C01818=1103.978,373.015,-89.633,-179.779,17.252,151.645
C01819=1103.984,373.262,-89.668,-179.776,17.255,151.645
C01820=1103.989,373.509,-89.704,-179.773,17.259,151.646
C01821=1103.995,373.757,-89.740,-179.770,17.264,151.646
C01822=1104.002,374.004,-89.776,-179.768,17.268,151.646
C01823=1104.007,374.251,-89.811,-179.765,17.272,151.647
C01824=1104.012,374.499,-89.848,-179.762,17.276,151.647
C01825=1104.018,374.745,-89.884,-179.760,17.280,151.648
C01826=1104.024,374.993,-89.919,-179.757,17.284,151.648
C01827=1104.029,375.240,-89.955,-179.754,17.289,151.649
C01828=1104.035,375.487,-89.992,-179.751,17.293,151.649
C01829=1104.041,375.735,-90.028,-179.748,17.297,151.650
C01830=1104.046,375.982,-90.064,-179.746,17.302,151.650
C01831=1104.052,376.229,-90.100,-179.743,17.306,151.651
C01832=1104.058,376.476,-90.135,-179.740,17.310,151.651
C01833=1104.063,376.724,-90.172,-179.737,17.314,151.652
C01834=1104.069,376.971,-90.208,-179.735,17.319,151.653
C01835=1104.075,377.218,-90.244,-179.732,17.323,151.653
C01836=1104.080,377.466,-90.281,-179.728,17.328,151.653
C01837=1104.086,377.713,-90.316,-179.727,17.332,151.654
C01838=1104.092,377.960,-90.352,-179.724,17.336,151.655
C01839=1104.097,378.208,-90.389,-179.721,17.341,151.655
C01840=1104.103,378.454,-90.425,-179.718,17.345,151.656
C01841=1104.108,378.702,-90.461,-179.716,17.349,151.656
C01842=1104.115,378.949,-90.498,-179.713,17.354,151.657
C01843=1104.120,379.195,-90.534,-179.710,17.358,151.657
C01844=1104.126,379.443,-90.570,-179.707,17.363,151.658
C01845=1104.132,379.690,-90.606,-179.704,17.368,151.659
C01846=1104.137,379.938,-90.643,-179.702,17.372,151.659
C01847=1104.143,380.185,-90.679,-179.699,17.376,151.660
C01848=1104.149,380.432,-90.716,-179.696,17.381,151.660
C01849=1104.155,380.680,-90.752,-179.694,17.385,151.661
C01850=1104.160,380.927,-90.788,-179.691,17.390,151.661
C01851=1104.166,381.174,-90.825,-179.689,17.394,151.662
C01852=1104.171,381.422,-90.861,-179.686,17.399,151.663
C01853=1104.178,381.669,-90.897,-179.683,17.404,151.663
C01854=1104.183,381.915,-90.934,-179.680,17.408,151.664
C01855=1104.189,382.162,-90.971,-179.678,17.413,151.664
C01856=1104.195,382.410,-91.008,-179.674,17.417,151.665
C01857=1104.201,382.657,-91.043,-179.673,17.422,151.666
C01858=1104.210,383.071,-91.105,-179.668,17.430,151.667
C01859=1104.219,383.485,-91.166,-179.663,17.438,151.668
C01860=1104.228,383.899,-91.227,-179.659,17.446,151.669
C01861=1104.239,384.314,-91.289,-179.655,17.454,151.670
C01862=1104.244,384.561,-91.326,-179.652,17.458,151.671
C01863=1104.249,384.808,-91.363,-179.649,17.463,151.671
C01864=1104.256,385.055,-91.399,-179.647,17.468,151.672
C01865=1104.261,385.302,-91.436,-179.644,17.473,151.673
C01866=1104.266,385.549,-91.473,-179.641,17.478,151.673
C01867=1104.273,385.796,-91.509,-179.639,17.483,151.674
C01868=1104.278,386.043,-91.546,-179.636,17.488,151.675
C01869=1104.284,386.291,-91.583,-179.634,17.493,151.676
C01870=1104.289,386.537,-91.620,-179.631,17.498,151.676
C01871=1104.295,386.785,-91.657,-179.629,17.502,151.677
C01872=1104.301,387.032,-91.694,-179.626,17.507,151.678
C01873=1104.306,387.279,-91.731,-179.624,17.512,151.678
C01874=1104.312,387.526,-91.768,-179.621,17.517,151.679
C01875=1104.318,387.773,-91.805,-179.619,17.522,151.680
C01876=1104.324,388.020,-91.841,-179.616,17.527,151.681
C01877=1104.329,388.267,-91.879,-179.613,17.532,151.681
C01878=1104.335,388.514,-91.916,-179.611,17.537,151.682
C01879=1104.340,388.762,-91.953,-179.609,17.542,151.683
C01880=1104.346,389.009,-91.990,-179.606,17.547,151.684
C01881=1104.353,389.256,-92.027,-179.603,17.552,151.684
C01882=1104.358,389.503,-92.064,-179.601,17.557,151.685
C01883=1104.364,389.750,-92.101,-179.598,17.563,151.686
C01884=1104.369,389.996,-92.138,-179.596,17.568,151.687
C01885=1104.375,390.244,-92.175,-179.593,17.573,151.687
C01886=1104.380,390.491,-92.212,-179.591,17.578,151.688
C01887=1104.386,390.738,-92.250,-179.588,17.583,151.689
C01888=1104.393,390.985,-92.287,-179.586,17.588,151.690
C01889=1104.398,391.232,-92.324,-179.583,17.593,151.690
C01890=1104.404,391.479,-92.361,-179.581,17.599,151.691
C01891=1104.410,391.726,-92.398,-179.578,17.604,151.692
C01892=1104.415,391.974,-92.435,-179.576,17.609,151.693
C01893=1104.421,392.220,-92.473,-179.573,17.615,151.694
C01894=1104.427,392.468,-92.510,-179.570,17.620,151.695
C01895=1104.433,392.715,-92.548,-179.568,17.625,151.695
C01896=1104.438,392.962,-92.585,-179.565,17.631,151.696
C01897=1104.444,393.209,-92.623,-179.563,17.636,151.697
C01898=1104.450,393.456,-92.660,-179.561,17.641,151.698
C01899=1104.456,393.703,-92.698,-179.558,17.646,151.699
C01900=1104.461,393.950,-92.735,-179.556,17.652,151.700
C01901=1104.467,394.197,-92.772,-179.553,17.657,151.701
C01902=1104.473,394.444,-92.809,-179.551,17.663,151.702
C01903=1104.479,394.691,-92.847,-179.549,17.668,151.703
C01904=1104.483,394.939,-92.885,-179.547,17.673,151.703
C01905=1104.489,395.185,-92.923,-179.544,17.679,151.704
C01906=1104.495,395.432,-92.960,-179.541,17.685,151.705
C01907=1104.501,395.680,-92.997,-179.539,17.690,151.706
C01908=1104.507,395.926,-93.035,-179.537,17.696,151.707
C01909=1104.513,396.173,-93.073,-179.534,17.701,151.708
C01910=1104.518,396.387,-93.105,-179.533,17.706,151.709
C01911=1104.523,396.600,-93.138,-179.530,17.711,151.709
C01912=1104.528,396.813,-93.170,-179.529,17.716,151.710
C01913=1104.533,397.026,-93.203,-179.526,17.721,151.711
C01914=1104.537,397.239,-93.236,-179.524,17.725,151.712
C01915=1104.542,397.453,-93.269,-179.522,17.731,151.713
C01916=1104.547,397.666,-93.301,-179.520,17.735,151.714
C01917=1104.552,397.879,-93.334,-179.518,17.741,151.714
C01918=1104.557,398.126,-93.371,-179.516,17.746,151.715
C01919=1104.563,398.373,-93.408,-179.513,17.752,151.716
C01920=1104.569,398.621,-93.447,-179.511,17.757,151.717
C01921=1104.575,398.868,-93.485,-179.509,17.763,151.718
C01922=1104.581,399.114,-93.523,-179.506,17.769,151.719
C01923=1104.586,399.361,-93.560,-179.504,17.775,151.720
C01924=1104.592,399.608,-93.599,-179.502,17.781,151.721
C01925=1104.597,399.855,-93.636,-179.500,17.786,151.722
C01926=1104.604,400.103,-93.674,-179.497,17.793,151.723
C01927=1104.609,400.350,-93.712,-179.495,17.798,151.724
C01928=1104.615,400.597,-93.750,-179.493,17.804,151.725
C01929=1104.620,400.844,-93.788,-179.491,17.810,151.727
C01930=1104.626,401.090,-93.826,-179.488,17.816,151.728
C01931=1104.631,401.338,-93.864,-179.486,17.822,151.729
C01932=1104.638,401.585,-93.902,-179.484,17.828,151.730
C01933=1104.643,401.832,-93.940,-179.482,17.834,151.731
C01934=1104.649,402.079,-93.979,-179.479,17.840,151.732
C01935=1104.655,402.326,-94.016,-179.477,17.846,151.733
C01936=1104.660,402.573,-94.055,-179.475,17.852,151.734
C01937=1104.666,402.820,-94.093,-179.472,17.859,151.735
C01938=1104.671,403.067,-94.131,-179.470,17.865,151.736
C01939=1104.678,403.313,-94.170,-179.468,17.871,151.737
C01940=1104.683,403.560,-94.208,-179.465,17.877,151.738
C01941=1104.689,403.808,-94.246,-179.463,17.883,151.739
C01942=1104.694,404.055,-94.284,-179.462,17.889,151.741
C01943=1104.700,404.302,-94.322,-179.459,17.896,151.742
C01944=1104.706,404.549,-94.361,-179.457,17.902,151.743
C01945=1104.712,404.796,-94.400,-179.455,17.908,151.744
C01946=1104.717,405.042,-94.438,-179.453,17.915,151.745
C01947=1104.723,405.290,-94.476,-179.451,17.921,151.746
C01948=1104.729,405.537,-94.514,-179.448,17.928,151.748
C01949=1104.735,405.783,-94.553,-179.446,17.933,151.749
C01950=1104.740,406.030,-94.592,-179.444,17.940,151.750
C01951=1104.746,406.277,-94.629,-179.442,17.946,151.751
C01952=1104.752,406.524,-94.669,-179.440,17.953,151.752
C01953=1104.757,406.771,-94.707,-179.437,17.960,151.754
C01954=1104.763,407.018,-94.745,-179.435,17.965,151.755
C01955=1104.769,407.265,-94.784,-179.433,17.972,151.756
C01956=1104.774,407.512,-94.823,-179.431,17.979,151.757
C01957=1104.780,407.758,-94.861,-179.429,17.986,151.758
C01958=1104.786,408.006,-94.900,-179.427,17.992,151.760
C01959=1104.791,408.253,-94.938,-179.424,17.999,151.761
C01960=1104.797,408.500,-94.977,-179.423,18.005,151.762
C01961=1104.802,408.747,-95.016,-179.420,18.012,151.763
C01962=1104.809,408.994,-95.055,-179.418,18.018,151.765
C01963=1104.814,409.241,-95.093,-179.416,18.026,151.766
C01964=1104.820,409.488,-95.132,-179.414,18.032,151.767
C01965=1104.825,409.735,-95.171,-179.412,18.039,151.769
C01966=1104.830,409.948,-95.205,-179.410,18.045,151.770
C01967=1104.835,410.161,-95.238,-179.408,18.051,151.771
C01968=1104.840,410.374,-95.272,-179.407,18.056,151.772
C01969=1104.845,410.587,-95.304,-179.405,18.062,151.773
C01970=1104.849,410.800,-95.338,-179.403,18.068,151.774
C01971=1104.854,411.013,-95.372,-179.401,18.074,151.775
C01972=1104.860,411.226,-95.405,-179.399,18.080,151.776
C01973=1104.864,411.439,-95.439,-179.398,18.086,151.778
C01974=1104.869,411.686,-95.478,-179.395,18.093,151.779
C01975=1104.876,411.933,-95.517,-179.393,18.100,151.780
C01976=1104.882,412.179,-95.556,-179.392,18.107,151.782
C01977=1104.888,412.426,-95.595,-179.389,18.114,151.783
C01978=1104.893,412.673,-95.633,-179.387,18.121,151.784
C01979=1104.899,412.921,-95.673,-179.385,18.128,151.786
C01980=1104.905,413.167,-95.712,-179.383,18.135,151.787
C01981=1104.911,413.414,-95.751,-179.381,18.142,151.789
C01982=1104.916,413.661,-95.790,-179.379,18.149,151.790
C01983=1104.922,413.908,-95.829,-179.377,18.156,151.791
C01984=1104.927,414.155,-95.868,-179.375,18.164,151.793
C01985=1104.933,414.402,-95.908,-179.374,18.171,151.794
C01986=1104.939,414.648,-95.947,-179.371,18.178,151.796
C01987=1104.945,414.896,-95.986,-179.369,18.185,151.797
C01988=1104.950,415.142,-96.025,-179.367,18.193,151.799
C01989=1104.956,415.389,-96.065,-179.365,18.200,151.800
C01990=1104.962,415.636,-96.104,-179.363,18.207,151.802
C01991=1104.968,415.883,-96.143,-179.361,18.215,151.803
C01992=1104.973,416.129,-96.182,-179.359,18.222,151.804
C01993=1104.980,416.376,-96.222,-179.358,18.229,151.806
C01994=1104.985,416.623,-96.261,-179.355,18.236,151.807
C01995=1104.991,416.870,-96.300,-179.353,18.244,151.809
C01996=1104.996,417.117,-96.340,-179.351,18.252,151.810
C01997=1105.002,417.364,-96.379,-179.349,18.259,151.812
C01998=1105.007,417.610,-96.418,-179.348,18.267,151.814
C01999=1105.014,417.857,-96.458,-179.346,18.274,151.815
C02000=1105.019,418.103,-96.498,-179.344,18.282,151.817
C02001=1105.025,418.351,-96.538,-179.342,18.290,151.818
C02002=1105.031,418.598,-96.577,-179.340,18.297,151.820
C02003=1105.036,418.844,-96.616,-179.338,18.305,151.821
C02004=1105.042,419.091,-96.656,-179.336,18.313,151.823
C02005=1105.047,419.337,-96.696,-179.334,18.321,151.825
C02006=1105.053,419.584,-96.735,-179.333,18.328,151.826
C02007=1105.059,419.831,-96.774,-179.331,18.336,151.828
C02008=1105.065,420.077,-96.815,-179.329,18.344,151.830
C02009=1105.071,420.325,-96.855,-179.327,18.352,151.831
C02010=1105.076,420.571,-96.894,-179.325,18.360,151.833
C02011=1105.082,420.818,-96.934,-179.323,18.368,151.834
C02012=1105.087,421.065,-96.973,-179.321,18.375,151.836
C02013=1105.093,421.312,-97.013,-179.319,18.383,151.838
C02014=1105.100,421.558,-97.053,-179.318,18.392,151.839
C02015=1105.104,421.805,-97.093,-179.316,18.400,151.841
C02016=1105.111,422.051,-97.133,-179.314,18.408,151.843
C02017=1105.117,422.299,-97.172,-179.312,18.416,151.844
C02018=1105.122,422.545,-97.213,-179.310,18.424,151.846
C02019=1105.128,422.792,-97.252,-179.308,18.432,151.848
C02020=1105.134,423.038,-97.292,-179.307,18.440,151.850
C02021=1105.139,423.285,-97.332,-179.305,18.448,151.851
C02022=1105.144,423.505,-97.368,-179.304,18.455,151.853
C02023=1105.150,423.724,-97.403,-179.302,18.463,151.854
C02024=1105.155,423.944,-97.439,-179.300,18.470,151.856
C02025=1105.160,424.164,-97.474,-179.299,18.477,151.858
C02026=1105.164,424.383,-97.510,-179.297,18.485,151.859
C02027=1105.169,424.604,-97.546,-179.296,18.492,151.861
C02028=1105.174,424.822,-97.582,-179.294,18.500,151.862
C02029=1105.179,425.043,-97.618,-179.293,18.507,151.864
C02030=1105.186,425.289,-97.658,-179.291,18.516,151.866
C02031=1105.191,425.536,-97.697,-179.290,18.524,151.868
C02032=1105.197,425.782,-97.738,-179.288,18.533,151.869
C02033=1105.203,426.029,-97.778,-179.286,18.542,151.871
C02034=1105.208,426.275,-97.818,-179.284,18.550,151.873
C02035=1105.214,426.523,-97.858,-179.282,18.559,151.875
C02036=1105.220,426.769,-97.898,-179.281,18.567,151.877
C02037=1105.226,427.016,-97.939,-179.279,18.576,151.879
C02038=1105.231,427.262,-97.979,-179.278,18.584,151.881
C02039=1105.237,427.509,-98.020,-179.277,18.593,151.883
C02040=1105.243,427.755,-98.060,-179.274,18.602,151.885
C02041=1105.249,428.002,-98.100,-179.273,18.611,151.886
C02042=1105.254,428.249,-98.140,-179.271,18.619,151.888
C02043=1105.260,428.495,-98.181,-179.270,18.628,151.890
C02044=1105.266,428.742,-98.221,-179.268,18.637,151.892
C02045=1105.272,428.989,-98.262,-179.266,18.646,151.894
C02046=1105.277,429.236,-98.302,-179.265,18.655,151.896
C02047=1105.283,429.481,-98.342,-179.263,18.664,151.898
C02048=1105.289,429.728,-98.383,-179.262,18.673,151.900
C02049=1105.294,429.975,-98.424,-179.260,18.682,151.902
C02050=1105.300,430.221,-98.465,-179.259,18.691,151.904
C02051=1105.306,430.467,-98.505,-179.257,18.700,151.906
C02052=1105.312,430.714,-98.546,-179.255,18.710,151.908
C02053=1105.317,430.961,-98.586,-179.254,18.719,151.910
C02054=1105.323,431.208,-98.627,-179.253,18.728,151.912
C02055=1105.329,431.454,-98.668,-179.251,18.737,151.914
C02056=1105.334,431.700,-98.708,-179.249,18.747,151.917
C02057=1105.340,431.946,-98.749,-179.248,18.756,151.919
C02058=1105.346,432.193,-98.790,-179.247,18.765,151.921
C02059=1105.352,432.440,-98.831,-179.245,18.775,151.923
C02060=1105.357,432.687,-98.871,-179.244,18.784,151.925
C02061=1105.363,432.933,-98.913,-179.243,18.793,151.927
C02062=1105.368,433.179,-98.953,-179.241,18.803,151.929
C02063=1105.375,433.426,-98.993,-179.240,18.812,151.931
C02064=1105.381,433.672,-99.035,-179.238,18.822,151.934
C02065=1105.386,433.919,-99.076,-179.237,18.832,151.936
C02066=1105.392,434.166,-99.116,-179.236,18.841,151.938
C02067=1105.398,434.412,-99.158,-179.234,18.851,151.940
C02068=1105.403,434.659,-99.198,-179.233,18.861,151.943
C02069=1105.408,434.904,-99.240,-179.231,18.870,151.945
C02070=1105.414,435.151,-99.281,-179.230,18.880,151.947
C02071=1105.419,435.398,-99.322,-179.229,18.890,151.949
C02072=1105.425,435.644,-99.363,-179.228,18.900,151.951
C02073=1105.431,435.891,-99.404,-179.226,18.910,151.954
C02074=1105.437,436.137,-99.445,-179.225,18.919,151.956
C02075=1105.443,436.384,-99.487,-179.224,18.930,151.958
C02076=1105.448,436.630,-99.528,-179.223,18.940,151.961
C02077=1105.454,436.877,-99.569,-179.221,18.950,151.963
C02078=1105.459,437.090,-99.605,-179.220,18.958,151.965
C02079=1105.464,437.303,-99.640,-179.219,18.967,151.967
C02080=1105.468,437.516,-99.676,-179.219,18.976,151.969
C02081=1105.474,437.731,-99.712,-179.217,18.985,151.971
C02082=1105.479,437.944,-99.747,-179.216,18.994,151.973
C02083=1105.484,438.157,-99.784,-179.215,19.002,151.975
C02084=1105.489,438.371,-99.819,-179.214,19.011,151.977
C02085=1105.494,438.584,-99.855,-179.213,19.020,151.979
C02086=1105.500,438.831,-99.896,-179.212,19.030,151.982
C02087=1105.506,439.077,-99.937,-179.210,19.041,151.984
C02088=1105.511,439.324,-99.979,-179.209,19.052,151.987
C02089=1105.517,439.570,-100.020,-179.208,19.062,151.989
C02090=1105.523,439.816,-100.062,-179.207,19.072,151.992
C02091=1105.529,440.062,-100.103,-179.206,19.083,151.994
C02092=1105.535,440.309,-100.145,-179.205,19.093,151.997
C02093=1105.539,440.556,-100.186,-179.204,19.104,151.999
C02094=1105.545,440.802,-100.228,-179.203,19.114,152.002
C02095=1105.551,441.048,-100.269,-179.202,19.125,152.004
C02096=1105.557,441.294,-100.311,-179.200,19.136,152.007
C02097=1105.562,441.541,-100.353,-179.200,19.147,152.009
C02098=1105.568,441.787,-100.394,-179.199,19.158,152.012
C02099=1105.574,442.033,-100.436,-179.197,19.169,152.014
C02100=1105.580,442.280,-100.478,-179.197,19.179,152.017
C02101=1105.586,442.526,-100.519,-179.196,19.190,152.020
C02102=1105.591,442.772,-100.561,-179.195,19.202,152.022
C02103=1105.597,443.018,-100.603,-179.194,19.212,152.025
C02104=1105.603,443.264,-100.645,-179.193,19.223,152.028
C02105=1105.608,443.511,-100.687,-179.192,19.235,152.030
C02106=1105.614,443.757,-100.728,-179.191,19.245,152.033
C02107=1105.620,444.004,-100.771,-179.190,19.257,152.036
C02108=1105.626,444.250,-100.812,-179.190,19.268,152.039
C02109=1105.631,444.497,-100.854,-179.190,19.278,152.041
C02110=1105.637,444.743,-100.896,-179.190,19.290,152.044
C02111=1105.643,444.989,-100.938,-179.190,19.301,152.047
C02112=1105.648,445.235,-100.980,-179.190,19.312,152.050
C02113=1105.654,445.482,-101.022,-179.190,19.323,152.053
C02114=1105.660,445.727,-101.064,-179.190,19.333,152.055
C02115=1105.666,445.975,-101.106,-179.190,19.345,152.058
C02116=1105.672,446.221,-101.148,-179.191,19.355,152.061
C02117=1105.677,446.467,-101.190,-179.192,19.366,152.064
C02118=1105.683,446.713,-101.232,-179.192,19.377,152.067
C02119=1105.688,446.959,-101.274,-179.193,19.388,152.070
C02120=1105.694,447.206,-101.316,-179.194,19.399,152.073
C02121=1105.700,447.452,-101.358,-179.195,19.410,152.076
C02122=1105.706,447.699,-101.401,-179.197,19.421,152.079
C02123=1105.711,447.945,-101.443,-179.198,19.432,152.082
C02124=1105.717,448.191,-101.485,-179.199,19.443,152.085
C02125=1105.722,448.437,-101.527,-179.201,19.453,152.088
C02126=1105.728,448.683,-101.570,-179.201,19.464,152.091
C02127=1105.734,448.930,-101.612,-179.203,19.475,152.094
C02128=1105.740,449.177,-101.654,-179.205,19.486,152.097
C02129=1105.745,449.423,-101.697,-179.207,19.496,152.100
C02130=1105.751,449.669,-101.738,-179.209,19.507,152.103
C02131=1105.757,449.915,-101.781,-179.211,19.517,152.106
C02132=1105.762,450.162,-101.823,-179.213,19.529,152.109
C02133=1105.769,450.407,-101.865,-179.215,19.539,152.112
C02134=1105.364,450.401,-101.989,-179.292,19.769,152.185
C02135=1105.357,450.155,-101.947,-179.290,19.758,152.182
C02136=1105.352,449.909,-101.905,-179.288,19.747,152.179
C02137=1105.346,449.662,-101.862,-179.286,19.736,152.175
C02138=1105.340,449.416,-101.820,-179.284,19.726,152.172
C02139=1105.335,449.170,-101.778,-179.283,19.715,152.169
C02140=1105.329,448.924,-101.735,-179.282,19.704,152.166
C02141=1105.323,448.678,-101.693,-179.280,19.693,152.163
C02142=1105.317,448.431,-101.651,-179.278,19.682,152.160
C02143=1105.312,448.185,-101.608,-179.277,19.671,152.157
C02144=1105.307,447.938,-101.566,-179.275,19.661,152.154
C02145=1105.301,447.692,-101.525,-179.274,19.649,152.151
C02146=1105.294,447.446,-101.481,-179.273,19.638,152.148
C02147=1105.289,447.199,-101.439,-179.273,19.627,152.145
C02148=1105.283,446.953,-101.397,-179.272,19.616,152.142
C02149=1105.278,446.707,-101.355,-179.271,19.605,152.139
C02150=1105.273,446.460,-101.313,-179.270,19.594,152.136
C02151=1105.266,446.215,-101.271,-179.269,19.583,152.133
C02152=1105.260,445.968,-101.229,-179.269,19.572,152.130
C02153=1105.255,445.721,-101.187,-179.268,19.561,152.127
C02154=1105.249,445.476,-101.144,-179.269,19.550,152.125
C02155=1105.243,445.229,-101.103,-179.268,19.539,152.122
C02156=1105.238,444.983,-101.061,-179.268,19.528,152.119
C02157=1105.231,444.737,-101.018,-179.268,19.517,152.116
C02158=1105.226,444.490,-100.976,-179.268,19.506,152.113
C02159=1105.220,444.244,-100.935,-179.269,19.495,152.111
C02160=1105.215,443.997,-100.893,-179.270,19.483,152.108
C02161=1105.208,443.752,-100.851,-179.270,19.473,152.105
C02162=1105.203,443.505,-100.808,-179.271,19.461,152.102
C02163=1105.197,443.259,-100.767,-179.272,19.450,152.100
C02164=1105.192,443.013,-100.725,-179.273,19.439,152.097
C02165=1105.186,442.766,-100.684,-179.274,19.428,152.094
C02166=1105.181,442.520,-100.641,-179.274,19.417,152.092
C02167=1105.174,442.274,-100.599,-179.276,19.406,152.089
C02168=1105.168,442.027,-100.557,-179.277,19.395,152.086
C02169=1105.163,441.781,-100.515,-179.278,19.383,152.084
C02170=1105.157,441.535,-100.474,-179.279,19.373,152.081
C02171=1105.151,441.288,-100.433,-179.280,19.362,152.079
C02172=1105.146,441.042,-100.390,-179.281,19.351,152.076
C02173=1105.140,440.796,-100.349,-179.282,19.340,152.074
C02174=1105.134,440.549,-100.308,-179.283,19.329,152.071
C02175=1105.129,440.303,-100.265,-179.285,19.319,152.068
C02176=1105.123,440.057,-100.224,-179.286,19.309,152.066
C02177=1105.117,439.811,-100.183,-179.287,19.298,152.064
C02178=1105.111,439.564,-100.141,-179.288,19.287,152.061
C02179=1105.105,439.318,-100.100,-179.289,19.277,152.059
C02180=1105.100,439.071,-100.058,-179.291,19.266,152.056
C02181=1105.094,438.825,-100.017,-179.291,19.256,152.054
C02182=1105.088,438.579,-99.975,-179.293,19.245,152.051
C02183=1105.083,438.367,-99.940,-179.294,19.236,152.049
C02184=1105.078,438.156,-99.904,-179.295,19.228,152.047
C02185=1105.073,437.945,-99.869,-179.296,19.218,152.045
C02186=1105.068,437.733,-99.833,-179.297,19.210,152.043
C02187=1105.063,437.522,-99.798,-179.298,19.201,152.041
C02188=1105.058,437.311,-99.763,-179.300,19.192,152.039
C02189=1105.054,437.100,-99.728,-179.300,19.184,152.037
C02190=1105.048,436.889,-99.691,-179.302,19.175,152.035
C02191=1105.042,436.642,-99.651,-179.303,19.165,152.033
C02192=1105.037,436.396,-99.610,-179.304,19.154,152.030
C02193=1105.031,436.149,-99.569,-179.305,19.145,152.028
C02194=1105.025,435.903,-99.527,-179.307,19.134,152.026
C02195=1105.017,435.527,-99.464,-179.309,19.119,152.022
C02196=1105.008,435.152,-99.402,-179.311,19.104,152.019
C02197=1104.999,434.776,-99.338,-179.313,19.089,152.015
C02198=1104.991,434.401,-99.276,-179.315,19.074,152.012
C02199=1104.985,434.154,-99.235,-179.317,19.064,152.009
C02200=1104.979,433.908,-99.195,-179.318,19.055,152.007
C02201=1104.974,433.662,-99.154,-179.320,19.045,152.005
C02202=1104.968,433.415,-99.113,-179.321,19.035,152.003
C02203=1104.962,433.169,-99.071,-179.322,19.026,152.001
C02204=1104.957,432.922,-99.031,-179.324,19.016,151.999
C02205=1104.951,432.675,-98.990,-179.325,19.007,151.996
C02206=1104.944,432.430,-98.949,-179.327,18.997,151.994
C02207=1104.939,432.183,-98.908,-179.328,18.988,151.992
C02208=1104.933,431.936,-98.867,-179.329,18.978,151.990
C02209=1104.928,431.690,-98.827,-179.332,18.969,151.988
C02210=1104.922,431.444,-98.786,-179.333,18.959,151.986
C02211=1104.917,431.197,-98.745,-179.334,18.950,151.984
C02212=1104.911,430.950,-98.704,-179.336,18.941,151.982
C02213=1104.905,430.703,-98.664,-179.337,18.932,151.980
C02214=1104.899,430.457,-98.624,-179.339,18.922,151.978
C02215=1104.894,430.211,-98.582,-179.340,18.914,151.976
C02216=1104.888,429.964,-98.541,-179.342,18.904,151.973
C02217=1104.882,429.717,-98.501,-179.344,18.895,151.971
C02218=1104.876,429.471,-98.461,-179.345,18.886,151.970
C02219=1104.871,429.225,-98.420,-179.347,18.876,151.967
C02220=1104.865,428.978,-98.379,-179.348,18.868,151.965
C02221=1104.859,428.731,-98.339,-179.350,18.859,151.963
C02222=1104.853,428.485,-98.299,-179.351,18.850,151.961
C02223=1104.848,428.238,-98.258,-179.353,18.841,151.960
C02224=1104.841,427.991,-98.218,-179.355,18.832,151.958
C02225=1104.836,427.745,-98.177,-179.357,18.823,151.956
C02226=1104.830,427.498,-98.137,-179.358,18.814,151.954
C02227=1104.824,427.252,-98.096,-179.360,18.806,151.952
C02228=1104.818,427.005,-98.056,-179.361,18.797,151.950
C02229=1104.813,426.759,-98.016,-179.364,18.788,151.948
C02230=1104.807,426.512,-97.976,-179.365,18.779,151.946
C02231=1104.802,426.265,-97.935,-179.367,18.771,151.944
C02232=1104.795,426.018,-97.895,-179.368,18.762,151.942
C02233=1104.790,425.772,-97.855,-179.370,18.754,151.941
C02234=1104.784,425.526,-97.814,-179.372,18.745,151.939
C02235=1104.779,425.278,-97.774,-179.374,18.736,151.937
C02236=1104.773,425.031,-97.734,-179.376,18.728,151.935
C02237=1104.767,424.786,-97.694,-179.377,18.719,151.933
C02238=1104.761,424.539,-97.653,-179.379,18.711,151.931
C02239=1104.754,424.228,-97.603,-179.381,18.700,151.929
C02240=1104.747,423.917,-97.553,-179.383,18.690,151.927
C02241=1104.740,423.607,-97.502,-179.386,18.679,151.925
C02242=1104.733,423.296,-97.452,-179.387,18.669,151.922
C02243=1104.727,423.050,-97.412,-179.389,18.661,151.921
C02244=1104.721,422.802,-97.372,-179.392,18.652,151.919
C02245=1104.715,422.556,-97.332,-179.393,18.644,151.917
C02246=1104.710,422.309,-97.292,-179.395,18.636,151.915
C02247=1104.704,422.063,-97.252,-179.397,18.627,151.914
C02248=1104.698,421.816,-97.212,-179.399,18.619,151.912
C02249=1104.693,421.569,-97.172,-179.401,18.611,151.910
C02250=1104.687,421.322,-97.133,-179.403,18.603,151.909
C02251=1104.680,421.076,-97.092,-179.404,18.596,151.907
C02252=1104.676,420.829,-97.053,-179.406,18.588,151.905
C02253=1104.670,420.582,-97.013,-179.408,18.580,151.904
C02254=1104.664,420.336,-96.974,-179.410,18.572,151.902
C02255=1104.658,420.089,-96.934,-179.411,18.564,151.900
C02256=1104.652,419.842,-96.893,-179.414,18.556,151.899
C02257=1104.647,419.596,-96.854,-179.415,18.548,151.897
C02258=1104.641,419.349,-96.815,-179.417,18.540,151.895
C02259=1104.636,419.102,-96.775,-179.419,18.532,151.894
C02260=1104.629,418.855,-96.735,-179.421,18.524,151.892
C02261=1104.623,418.608,-96.696,-179.423,18.517,151.891
C02262=1104.618,418.362,-96.657,-179.425,18.508,151.889
C02263=1104.613,418.114,-96.617,-179.427,18.501,151.887
C02264=1104.607,417.869,-96.577,-179.429,18.494,151.886
C02265=1104.601,417.621,-96.537,-179.431,18.486,151.884
C02266=1104.595,417.375,-96.498,-179.433,18.478,151.883
C02267=1104.589,417.128,-96.459,-179.435,18.470,151.881
C02268=1104.584,416.881,-96.419,-179.437,18.463,151.880
C02269=1104.578,416.634,-96.380,-179.439,18.455,151.878
C02270=1104.572,416.387,-96.340,-179.440,18.448,151.877
C02271=1104.567,416.140,-96.301,-179.443,18.441,151.875
C02272=1104.561,415.893,-96.262,-179.445,18.433,151.874
C02273=1104.555,415.647,-96.222,-179.447,18.425,151.872
C02274=1104.549,415.400,-96.183,-179.448,18.419,151.871
C02275=1104.543,415.154,-96.144,-179.451,18.411,151.869
C02276=1104.537,414.907,-96.104,-179.453,18.404,151.868
C02277=1104.532,414.660,-96.066,-179.455,18.396,151.866
C02278=1104.526,414.412,-96.026,-179.457,18.389,151.865
C02279=1104.521,414.166,-95.987,-179.459,18.382,151.863
C02280=1104.515,413.919,-95.948,-179.461,18.374,151.862
C02281=1104.509,413.672,-95.909,-179.463,18.367,151.861
C02282=1104.503,413.425,-95.869,-179.465,18.360,151.859
C02283=1104.498,413.179,-95.830,-179.467,18.353,151.858
C02284=1104.491,412.932,-95.791,-179.469,18.345,151.856
C02285=1104.486,412.685,-95.753,-179.471,18.339,151.855
C02286=1104.480,412.438,-95.713,-179.473,18.331,151.854
C02287=1104.475,412.191,-95.674,-179.476,18.324,151.852
C02288=1104.469,411.944,-95.635,-179.477,18.318,151.851
C02289=1104.463,411.698,-95.596,-179.479,18.310,151.849
C02290=1104.457,411.450,-95.557,-179.482,18.303,151.848
C02291=1104.452,411.237,-95.523,-179.483,18.298,151.847
C02292=1104.447,411.024,-95.490,-179.485,18.291,151.846
C02293=1104.442,410.811,-95.456,-179.487,18.285,151.845
C02294=1104.437,410.597,-95.423,-179.489,18.279,151.843
C02295=1104.433,410.384,-95.389,-179.491,18.273,151.842
C02296=1104.428,410.171,-95.355,-179.493,18.267,151.841
C02297=1104.423,409.957,-95.322,-179.495,18.261,151.840
C02298=1104.418,409.744,-95.288,-179.496,18.256,151.839
C02299=1104.412,409.498,-95.249,-179.498,18.249,151.838
C02300=1104.407,409.250,-95.211,-179.500,18.242,151.836
C02301=1104.401,409.004,-95.172,-179.502,18.235,151.835
C02302=1104.396,408.757,-95.133,-179.505,18.228,151.834
C02303=1104.389,408.510,-95.094,-179.507,18.222,151.832
C02304=1104.384,408.263,-95.056,-179.509,18.215,151.831
C02305=1104.379,408.016,-95.017,-179.511,18.208,151.830
C02306=1104.373,407.769,-94.978,-179.513,18.201,151.829
C02307=1104.367,407.522,-94.940,-179.515,18.195,151.827
C02308=1104.361,407.275,-94.901,-179.518,18.188,151.826
C02309=1104.355,407.028,-94.862,-179.520,18.182,151.825
C02310=1104.350,406.781,-94.824,-179.522,18.175,151.824
C02311=1104.344,406.534,-94.786,-179.524,18.169,151.822
C02312=1104.338,406.287,-94.746,-179.527,18.162,151.821
C02313=1104.333,406.040,-94.708,-179.528,18.155,151.820
C02314=1104.327,405.794,-94.670,-179.530,18.150,151.819
C02315=1104.321,405.546,-94.631,-179.533,18.143,151.818
C02316=1104.316,405.299,-94.593,-179.535,18.136,151.816
C02317=1104.310,405.053,-94.555,-179.538,18.130,151.815
C02318=1104.304,404.805,-94.515,-179.539,18.123,151.814
C02319=1104.298,404.559,-94.478,-179.542,18.117,151.813
C02320=1104.293,404.312,-94.439,-179.544,18.111,151.812
C02321=1104.287,404.065,-94.401,-179.546,18.105,151.811
C02322=1104.281,403.817,-94.363,-179.549,18.098,151.810
C02323=1104.276,403.571,-94.324,-179.551,18.092,151.808
C02324=1104.270,403.324,-94.286,-179.553,18.086,151.807
C02325=1104.264,403.076,-94.247,-179.555,18.080,151.806
C02326=1104.258,402.829,-94.209,-179.557,18.074,151.805
C02327=1104.253,402.582,-94.171,-179.559,18.068,151.804
C02328=1104.247,402.336,-94.133,-179.562,18.061,151.803
C02329=1104.242,402.089,-94.095,-179.564,18.055,151.802
C02330=1104.235,401.841,-94.057,-179.566,18.049,151.801
C02331=1104.230,401.594,-94.019,-179.569,18.042,151.799
C02332=1104.224,401.347,-93.981,-179.571,18.037,151.798
C02333=1104.218,401.101,-93.943,-179.573,18.031,151.797
C02334=1104.213,400.854,-93.905,-179.576,18.025,151.796
C02335=1104.207,400.606,-93.867,-179.578,18.019,151.795
C02336=1104.202,400.359,-93.828,-179.580,18.013,151.794
C02337=1104.196,400.112,-93.790,-179.582,18.007,151.793
C02338=1104.190,399.866,-93.753,-179.585,18.000,151.792
C02339=1104.185,399.619,-93.714,-179.587,17.995,151.791
C02340=1104.178,399.371,-93.676,-179.589,17.989,151.790
C02341=1104.172,399.124,-93.638,-179.591,17.983,151.789
C02342=1104.167,398.877,-93.600,-179.594,17.977,151.788
C02343=1104.161,398.631,-93.562,-179.597,17.971,151.787
C02344=1104.155,398.384,-93.525,-179.599,17.965,151.786
C02345=1104.150,398.136,-93.487,-179.601,17.960,151.785
C02346=1104.144,397.889,-93.449,-179.603,17.954,151.784
C02347=1104.139,397.676,-93.417,-179.605,17.949,151.783
C02348=1104.134,397.462,-93.384,-179.607,17.944,151.782
C02349=1104.129,397.249,-93.351,-179.609,17.939,151.781
C02350=1104.124,397.036,-93.319,-179.611,17.934,151.781
C02351=1104.120,396.822,-93.286,-179.614,17.929,151.780
C02352=1104.115,396.609,-93.253,-179.615,17.924,151.779
C02353=1104.110,396.396,-93.220,-179.618,17.919,151.778
C02354=1104.105,396.183,-93.188,-179.620,17.915,151.777
C02355=1104.099,395.935,-93.150,-179.622,17.909,151.776
C02356=1104.093,395.688,-93.113,-179.625,17.903,151.775
C02357=1104.087,395.441,-93.075,-179.627,17.897,151.775
C02358=1104.082,395.194,-93.037,-179.629,17.892,151.774
C02359=1104.076,394.947,-93.000,-179.632,17.886,151.773
C02360=1104.070,394.700,-92.962,-179.634,17.881,151.772
C02361=1104.065,394.453,-92.925,-179.636,17.875,151.771
C02362=1104.059,394.206,-92.887,-179.639,17.870,151.770
C02363=1104.053,393.959,-92.850,-179.641,17.865,151.769
C02364=1104.047,393.712,-92.813,-179.643,17.859,151.768
C02365=1104.041,393.465,-92.775,-179.647,17.853,151.767
C02366=1104.036,393.218,-92.738,-179.649,17.848,151.766
C02367=1104.030,392.971,-92.700,-179.651,17.842,151.766
C02368=1104.025,392.723,-92.662,-179.654,17.837,151.765
C02369=1104.019,392.477,-92.625,-179.656,17.832,151.764
C02370=1104.014,392.229,-92.588,-179.659,17.827,151.763
C02371=1104.007,391.982,-92.551,-179.661,17.821,151.762
C02372=1104.001,391.735,-92.513,-179.663,17.816,151.761
C02373=1103.996,391.488,-92.476,-179.666,17.811,151.761
C02374=1103.990,391.241,-92.439,-179.668,17.806,151.760
C02375=1103.984,390.994,-92.402,-179.671,17.801,151.759
C02376=1103.979,390.747,-92.364,-179.673,17.795,151.758
C02377=1103.973,390.500,-92.327,-179.676,17.790,151.757
C02378=1103.967,390.252,-92.290,-179.678,17.785,151.756
C02379=1103.962,390.005,-92.253,-179.681,17.780,151.756
C02380=1103.955,389.759,-92.215,-179.683,17.774,151.755
C02381=1103.950,389.512,-92.179,-179.686,17.769,151.754
C02382=1103.944,389.265,-92.142,-179.688,17.764,151.753
C02383=1103.938,389.018,-92.104,-179.691,17.759,151.753
C02384=1103.933,388.771,-92.067,-179.693,17.754,151.752
C02385=1103.927,388.523,-92.030,-179.696,17.749,151.751
C02386=1103.921,388.276,-91.993,-179.699,17.743,151.750
C02387=1103.915,388.029,-91.956,-179.702,17.738,151.750
C02388=1103.909,387.782,-91.919,-179.704,17.734,151.749
C02389=1103.904,387.535,-91.882,-179.706,17.729,151.748
C02390=1103.899,387.288,-91.845,-179.709,17.723,151.747
C02391=1103.892,387.041,-91.809,-179.712,17.719,151.747
C02392=1103.887,386.794,-91.771,-179.714,17.714,151.746
C02393=1103.881,386.546,-91.734,-179.717,17.708,151.745
C02394=1103.876,386.299,-91.697,-179.719,17.704,151.744
C02395=1103.870,386.052,-91.661,-179.722,17.699,151.744
C02396=1103.864,385.805,-91.624,-179.724,17.693,151.743
C02397=1103.859,385.558,-91.587,-179.727,17.689,151.742
C02398=1103.853,385.311,-91.550,-179.730,17.684,151.741
C02399=1103.847,385.064,-91.513,-179.733,17.679,151.741
C02400=1103.842,384.817,-91.477,-179.735,17.674,151.740
C02401=1103.836,384.569,-91.440,-179.738,17.669,151.739
C02402=1103.831,384.322,-91.403,-179.740,17.664,151.739
C02403=1103.821,383.908,-91.342,-179.745,17.656,151.738
C02404=1103.812,383.493,-91.280,-179.749,17.648,151.736
C02405=1103.802,383.079,-91.218,-179.754,17.640,151.735
C02406=1103.792,382.665,-91.157,-179.758,17.632,151.734
C02407=1103.786,382.417,-91.120,-179.761,17.627,151.734
C02408=1103.781,382.170,-91.085,-179.764,17.622,151.733
C02409=1103.775,381.923,-91.048,-179.766,17.618,151.732
C02410=1103.769,381.676,-91.011,-179.769,17.613,151.732
C02411=1103.763,381.429,-90.974,-179.771,17.609,151.731
C02412=1103.758,381.182,-90.939,-179.774,17.604,151.730
C02413=1103.752,380.934,-90.902,-179.777,17.599,151.730
C02414=1103.746,380.687,-90.865,-179.780,17.594,151.729
C02415=1103.740,380.440,-90.828,-179.782,17.590,151.729
C02416=1103.735,380.193,-90.793,-179.785,17.586,151.728
C02417=1103.729,379.945,-90.756,-179.788,17.581,151.727
C02418=1103.723,379.698,-90.719,-179.790,17.576,151.727
C02419=1103.718,379.451,-90.684,-179.793,17.572,151.726
C02420=1103.712,379.204,-90.647,-179.796,17.567,151.726
C02421=1103.706,378.956,-90.611,-179.798,17.563,151.725
C02422=1103.701,378.710,-90.575,-179.801,17.559,151.725
C02423=1103.695,378.463,-90.538,-179.804,17.554,151.724
C02424=1103.689,378.215,-90.502,-179.807,17.549,151.723
C02425=1103.684,377.968,-90.466,-179.810,17.545,151.723
C02426=1103.678,377.721,-90.430,-179.812,17.541,151.722
C02427=1103.672,377.473,-90.393,-179.815,17.536,151.722
C02428=1103.667,377.226,-90.358,-179.818,17.532,151.721
C02429=1103.661,376.979,-90.320,-179.821,17.527,151.721
C02430=1103.655,376.731,-90.285,-179.823,17.523,151.720
C02431=1103.649,376.484,-90.249,-179.826,17.519,151.720
C02432=1103.644,376.237,-90.212,-179.829,17.514,151.719
C02433=1103.638,375.990,-90.177,-179.832,17.510,151.719
C02434=1103.632,375.743,-90.141,-179.834,17.505,151.718
C02435=1103.627,375.495,-90.104,-179.837,17.501,151.717
C02436=1103.621,375.248,-90.069,-179.840,17.497,151.717
C02437=1103.615,375.001,-90.032,-179.843,17.493,151.717
C02438=1103.610,374.754,-89.996,-179.846,17.488,151.716
C02439=1103.604,374.506,-89.961,-179.848,17.484,151.715
C02440=1103.598,374.259,-89.924,-179.851,17.480,151.715
C02441=1103.593,374.012,-89.889,-179.854,17.475,151.714
C02442=1103.587,373.764,-89.853,-179.856,17.472,151.714
C02443=1103.582,373.517,-89.817,-179.859,17.467,151.714
C02444=1103.575,373.270,-89.781,-179.862,17.463,151.713
C02445=1103.569,373.022,-89.745,-179.865,17.459,151.713
C02446=1103.564,372.775,-89.710,-179.868,17.455,151.712
C02447=1103.558,372.528,-89.674,-179.871,17.451,151.712
C02448=1103.553,372.281,-89.639,-179.874,17.446,151.711
C02449=1103.546,372.034,-89.602,-179.876,17.443,151.711
C02450=1103.542,371.786,-89.566,-179.879,17.439,151.710
C02451=1103.536,371.539,-89.530,-179.882,17.434,151.710
C02452=1103.529,371.291,-89.495,-179.885,17.430,151.709
C02453=1103.524,371.044,-89.459,-179.888,17.426,151.709
C02454=1103.518,370.796,-89.424,-179.891,17.422,151.709
C02455=1103.509,370.409,-89.368,-179.895,17.416,151.708
C02456=1103.500,370.021,-89.312,-179.899,17.410,151.707
C02457=1103.491,369.633,-89.256,-179.904,17.404,151.707
C02458=1103.483,369.246,-89.201,-179.909,17.397,151.706
C02459=1103.477,368.999,-89.165,-179.911,17.393,151.706
C02460=1103.471,368.752,-89.129,-179.914,17.389,151.705
C02461=1103.465,368.504,-89.094,-179.917,17.385,151.705
C02462=1103.460,368.257,-89.059,-179.920,17.381,151.704
C02463=1103.454,368.009,-89.023,-179.923,17.377,151.704
C02464=1103.449,367.762,-88.988,-179.926,17.373,151.704
C02465=1103.443,367.514,-88.952,-179.929,17.370,151.703
C02466=1103.437,367.267,-88.917,-179.932,17.365,151.703
C02467=1103.431,367.020,-88.881,-179.934,17.362,151.702
C02468=1103.426,366.773,-88.846,-179.937,17.358,151.702
C02469=1103.421,366.525,-88.811,-179.940,17.354,151.702
C02470=1103.415,366.277,-88.775,-179.943,17.350,151.701
C02471=1103.409,366.030,-88.740,-179.946,17.346,151.701
C02472=1103.403,365.783,-88.704,-179.949,17.343,151.701
C02473=1103.398,365.535,-88.670,-179.952,17.339,151.700
C02474=1103.391,365.288,-88.635,-179.955,17.335,151.700
C02475=1103.386,365.041,-88.599,-179.958,17.331,151.700
C02476=1103.381,364.793,-88.565,-179.961,17.327,151.699
C02477=1103.375,364.546,-88.529,-179.964,17.324,151.699
C02478=1103.369,364.299,-88.493,-179.967,17.320,151.699
C02479=1103.363,364.051,-88.459,-179.969,17.316,151.698
C02480=1103.357,363.804,-88.424,-179.973,17.312,151.698
C02481=1103.351,363.556,-88.388,-179.975,17.309,151.698
C02482=1103.346,363.308,-88.353,-179.978,17.305,151.697
C02483=1103.341,363.061,-88.318,-179.982,17.301,151.697
C02484=1103.334,362.813,-88.283,-179.984,17.298,151.697
C02485=1103.329,362.566,-88.248,-179.988,17.294,151.696
C02486=1103.324,362.319,-88.213,-179.990,17.291,151.696
C02487=1103.318,362.071,-88.178,-179.994,17.287,151.696
C02488=1103.312,361.824,-88.144,-179.996,17.283,151.696
C02489=1103.306,361.576,-88.108,-180.000,17.280,151.695
C02490=1103.301,361.329,-88.073,179.998,17.276,151.695
C02491=1103.295,361.082,-88.039,179.995,17.272,151.695
C02492=1103.289,360.834,-88.004,179.992,17.269,151.694
C02493=1103.283,360.587,-87.968,179.989,17.265,151.694
C02494=1103.278,360.339,-87.934,179.986,17.262,151.694
C02495=1103.272,360.091,-87.899,179.983,17.258,151.694
C02496=1103.266,359.844,-87.864,179.980,17.255,151.693
C02497=1103.261,359.597,-87.830,179.977,17.251,151.693
C02498=1103.255,359.349,-87.794,179.974,17.248,151.693
C02499=1103.249,359.102,-87.759,179.970,17.244,151.693
C02500=1103.244,358.854,-87.725,179.968,17.241,151.692
C02501=1103.238,358.606,-87.690,179.965,17.237,151.692
C02502=1103.232,358.359,-87.655,179.962,17.234,151.692
C02503=1103.227,358.112,-87.621,179.958,17.230,151.692
C02504=1103.221,357.864,-87.587,179.956,17.227,151.691
C02505=1103.215,357.616,-87.552,179.952,17.223,151.691
C02506=1103.209,357.369,-87.517,179.949,17.220,151.691
C02507=1103.200,356.996,-87.464,179.945,17.215,151.691
C02508=1103.192,356.624,-87.413,179.941,17.210,151.690
C02509=1103.183,356.251,-87.361,179.936,17.205,151.690
C02510=1103.175,355.878,-87.308,179.931,17.200,151.690
C02511=1103.169,355.631,-87.274,179.928,17.197,151.689
C02512=1103.163,355.383,-87.239,179.925,17.193,151.689
C02513=1103.158,355.135,-87.205,179.922,17.190,151.689
C02514=1103.152,354.888,-87.171,179.919,17.187,151.689
C02515=1103.147,354.641,-87.137,179.916,17.183,151.689
C02516=1103.142,354.393,-87.102,179.913,17.180,151.688
C02517=1103.135,354.145,-87.067,179.910,17.176,151.688
C02518=1103.129,353.898,-87.033,179.907,17.173,151.688
C02519=1103.124,353.650,-86.999,179.903,17.170,151.688
C02520=1103.118,353.403,-86.965,179.900,17.167,151.688
C02521=1103.113,353.155,-86.930,179.898,17.164,151.688
C02522=1103.107,352.907,-86.896,179.894,17.160,151.687
C02523=1103.101,352.660,-86.862,179.891,17.157,151.687
C02524=1103.096,352.412,-86.827,179.888,17.153,151.687
C02525=1103.090,352.165,-86.793,179.885,17.151,151.687
C02526=1103.084,351.917,-86.760,179.882,17.148,151.687
C02527=1103.078,351.669,-86.725,179.879,17.144,151.687
C02528=1103.073,351.422,-86.690,179.876,17.141,151.686
C02529=1103.067,351.174,-86.656,179.873,17.138,151.686
C02530=1103.061,350.927,-86.622,179.869,17.135,151.686
C02531=1103.056,350.679,-86.588,179.867,17.132,151.686
C02532=1103.050,350.432,-86.554,179.863,17.128,151.686
C02533=1103.044,350.184,-86.520,179.860,17.126,151.686
C02534=1103.038,349.936,-86.486,179.857,17.123,151.686
C02535=1103.033,349.689,-86.451,179.854,17.119,151.685
C02536=1103.027,349.441,-86.418,179.851,17.116,151.685
C02537=1103.021,349.194,-86.384,179.848,17.113,151.685
C02538=1103.016,348.946,-86.350,179.844,17.110,151.685
C02539=1103.011,348.698,-86.316,179.841,17.107,151.685
C02540=1103.005,348.451,-86.282,179.838,17.104,151.685
C02541=1102.998,348.203,-86.247,179.835,17.101,151.685
C02542=1102.993,347.955,-86.214,179.832,17.098,151.685
C02543=1102.987,347.708,-86.180,179.829,17.095,151.685
C02544=1102.981,347.460,-86.146,179.825,17.092,151.684
C02545=1102.976,347.212,-86.112,179.823,17.089,151.684
C02546=1102.970,346.965,-86.078,179.820,17.086,151.684
C02547=1102.965,346.717,-86.045,179.816,17.083,151.684
C02548=1102.959,346.470,-86.011,179.813,17.080,151.684
C02549=1102.953,346.222,-85.977,179.810,17.077,151.684
C02550=1102.948,345.974,-85.943,179.807,17.074,151.684
C02551=1102.942,345.727,-85.910,179.804,17.071,151.684
C02552=1102.936,345.479,-85.876,179.800,17.068,151.684
C02553=1102.931,345.231,-85.842,179.798,17.065,151.684
C02554=1102.925,344.984,-85.808,179.794,17.062,151.684
C02555=1102.919,344.736,-85.775,179.791,17.059,151.683
C02556=1102.913,344.489,-85.741,179.788,17.056,151.683
C02557=1102.908,344.241,-85.708,179.785,17.054,151.683
C02558=1102.902,343.992,-85.674,179.781,17.050,151.683
C02559=1102.893,343.622,-85.623,179.777,17.046,151.683
C02560=1102.885,343.252,-85.573,179.772,17.042,151.683
C02561=1102.876,342.882,-85.523,179.767,17.038,151.683
C02562=1102.868,342.510,-85.472,179.762,17.034,151.683
C02563=1102.862,342.264,-85.440,179.760,17.031,151.683
C02564=1102.857,342.016,-85.406,179.756,17.028,151.683
C02565=1102.851,341.768,-85.373,179.753,17.025,151.683
C02566=1102.845,341.521,-85.339,179.750,17.022,151.683
C02567=1102.840,341.273,-85.306,179.747,17.020,151.683
C02568=1102.834,341.025,-85.272,179.743,17.017,151.683
C02569=1102.828,340.777,-85.239,179.740,17.014,151.683
C02570=1102.823,340.529,-85.206,179.737,17.011,151.683
C02571=1102.817,340.282,-85.172,179.734,17.009,151.683
C02572=1102.812,340.034,-85.138,179.730,17.005,151.683
C02573=1102.805,339.786,-85.105,179.727,17.003,151.683
C02574=1102.800,339.538,-85.072,179.724,17.000,151.683
C02575=1102.794,339.290,-85.039,179.721,16.997,151.683
C02576=1102.789,339.042,-85.005,179.718,16.995,151.683
C02577=1102.783,338.794,-84.972,179.714,16.992,151.683
C02578=1102.777,338.547,-84.939,179.711,16.989,151.683
C02579=1102.771,338.299,-84.906,179.708,16.987,151.683
C02580=1102.766,338.052,-84.873,179.705,16.984,151.683
C02581=1102.761,337.804,-84.840,179.702,16.982,151.683
C02582=1102.754,337.556,-84.807,179.698,16.979,151.683
C02583=1102.749,337.308,-84.774,179.695,16.976,151.683
C02584=1102.743,337.060,-84.740,179.692,16.973,151.683
C02585=1102.738,336.813,-84.707,179.688,16.971,151.683
C02586=1102.731,336.565,-84.674,179.685,16.968,151.683
C02587=1102.726,336.317,-84.641,179.682,16.966,151.683
C02588=1102.720,336.069,-84.608,179.678,16.963,151.683
C02589=1102.715,335.822,-84.575,179.675,16.960,151.683
C02590=1102.709,335.574,-84.542,179.672,16.958,151.683
C02591=1102.704,335.326,-84.509,179.669,16.955,151.683
C02592=1102.697,335.079,-84.476,179.666,16.953,151.683
C02593=1102.692,334.830,-84.443,179.663,16.950,151.683
C02594=1102.686,334.583,-84.410,179.659,16.948,151.683
C02595=1102.680,334.335,-84.377,179.656,16.945,151.683
C02596=1102.675,334.088,-84.344,179.653,16.942,151.683
C02597=1102.669,333.840,-84.311,179.649,16.940,151.683
C02598=1102.664,333.592,-84.279,179.646,16.938,151.683
C02599=1102.658,333.344,-84.245,179.643,16.935,151.683
C02600=1102.652,333.096,-84.213,179.640,16.933,151.683
C02601=1102.647,332.849,-84.180,179.637,16.930,151.683
C02602=1102.641,332.601,-84.148,179.633,16.927,151.683
C02603=1102.635,332.353,-84.114,179.629,16.925,151.684
C02604=1102.629,332.105,-84.082,179.626,16.922,151.684
C02605=1102.624,331.857,-84.049,179.623,16.920,151.684
C02606=1102.618,331.610,-84.017,179.620,16.918,151.684
C02607=1102.612,331.362,-83.983,179.617,16.915,151.684
C02608=1102.607,331.114,-83.951,179.613,16.913,151.684
C02609=1102.600,330.866,-83.918,179.610,16.910,151.684
C02610=1102.595,330.618,-83.885,179.607,16.908,151.684
C02611=1102.587,330.241,-83.836,179.602,16.905,151.684
C02612=1102.577,329.865,-83.787,179.597,16.900,151.684
C02613=1102.568,329.488,-83.737,179.592,16.897,151.685
C02614=1102.559,329.112,-83.687,179.587,16.894,151.685
C02615=1102.554,328.864,-83.656,179.583,16.892,151.685
C02616=1102.548,328.616,-83.622,179.580,16.889,151.685
C02617=1102.542,328.368,-83.590,179.577,16.887,151.685
C02618=1102.536,328.120,-83.558,179.574,16.884,151.685
C02619=1102.531,327.873,-83.525,179.570,16.882,151.685
C02620=1102.525,327.624,-83.493,179.567,16.880,151.685
C02621=1102.519,327.377,-83.461,179.564,16.878,151.685
C02622=1102.514,327.129,-83.429,179.561,16.876,151.686
C02623=1102.508,326.881,-83.396,179.556,16.873,151.686
C02624=1102.502,326.633,-83.364,179.553,16.870,151.686
C02625=1102.496,326.385,-83.332,179.550,16.868,151.686
C02626=1102.490,326.138,-83.299,179.546,16.866,151.686
C02627=1102.485,325.889,-83.267,179.543,16.864,151.686
C02628=1102.479,325.641,-83.235,179.540,16.861,151.686
C02629=1102.474,325.394,-83.203,179.537,16.859,151.687
C02630=1102.468,325.146,-83.170,179.534,16.857,151.687
C02631=1102.463,324.898,-83.138,179.530,16.855,151.687
C02632=1102.457,324.650,-83.106,179.527,16.853,151.687
C02633=1102.451,324.403,-83.073,179.524,16.850,151.687
C02634=1102.445,324.155,-83.042,179.520,16.848,151.687
C02635=1102.439,323.907,-83.010,179.517,16.846,151.687
C02636=1102.434,323.658,-82.977,179.513,16.844,151.688
C02637=1102.429,323.411,-82.945,179.510,16.842,151.688
C02638=1102.423,323.163,-82.913,179.507,16.839,151.688
C02639=1102.417,322.916,-82.881,179.504,16.837,151.688
C02640=1102.411,322.667,-82.849,179.500,16.835,151.688
C02641=1102.405,322.419,-82.817,179.497,16.833,151.688
C02642=1102.400,322.171,-82.785,179.494,16.830,151.688
C02643=1102.394,321.923,-82.752,179.490,16.828,151.688
C02644=1102.389,321.676,-82.721,179.487,16.826,151.689
C02645=1102.383,321.427,-82.689,179.484,16.824,151.689
C02646=1102.378,321.180,-82.657,179.480,16.822,151.689
C02647=1102.372,320.932,-82.625,179.477,16.820,151.689
C02648=1102.366,320.684,-82.593,179.473,16.818,151.689
C02649=1102.360,320.436,-82.561,179.470,16.815,151.689
C02650=1102.355,320.188,-82.530,179.467,16.813,151.690
C02651=1102.350,319.940,-82.497,179.464,16.811,151.690
C02652=1102.344,319.692,-82.465,179.460,16.809,151.690
C02653=1102.338,319.444,-82.433,179.457,16.807,151.690
C02654=1102.333,319.197,-82.402,179.453,16.805,151.690
C02655=1102.327,318.948,-82.370,179.450,16.802,151.691
C02656=1102.321,318.701,-82.338,179.447,16.800,151.691
C02657=1102.315,318.453,-82.306,179.443,16.798,151.691
C02658=1102.310,318.205,-82.274,179.441,16.797,151.691
C02659=1102.304,317.957,-82.242,179.437,16.795,151.691
C02660=1102.299,317.709,-82.211,179.434,16.793,151.691
C02661=1102.294,317.461,-82.180,179.431,16.790,151.691
C02662=1102.288,317.213,-82.148,179.427,16.788,151.692
C02663=1102.279,316.830,-82.099,179.422,16.785,151.692
C02664=1102.271,316.446,-82.050,179.416,16.781,151.692
C02665=1102.262,316.063,-82.001,179.411,16.778,151.693
C02666=1102.253,315.678,-81.951,179.406,16.775,151.693
C02667=1102.248,315.430,-81.920,179.403,16.773,151.693
C02668=1102.243,315.183,-81.889,179.399,16.771,151.693
C02669=1102.236,314.935,-81.857,179.397,16.769,151.693
C02670=1102.231,314.687,-81.826,179.393,16.767,151.694
C02671=1102.225,314.438,-81.794,179.390,16.766,151.694
C02672=1102.219,314.191,-81.763,179.386,16.763,151.694
C02673=1102.213,313.943,-81.731,179.383,16.761,151.694
C02674=1102.208,313.695,-81.700,179.379,16.760,151.695
C02675=1102.201,313.447,-81.669,179.376,16.758,151.695
C02676=1102.196,313.199,-81.638,179.372,16.756,151.695
C02677=1102.191,312.951,-81.606,179.369,16.754,151.695
C02678=1102.184,312.704,-81.575,179.365,16.752,151.696
C02679=1102.179,312.455,-81.544,179.362,16.751,151.696
C02680=1102.173,312.207,-81.512,179.359,16.748,151.696
C02681=1102.167,311.959,-81.482,179.356,16.746,151.696
C02682=1102.162,311.712,-81.450,179.352,16.745,151.697
C02683=1102.156,311.463,-81.419,179.348,16.743,151.697
C02684=1102.150,311.216,-81.387,179.345,16.741,151.697
C02685=1102.144,310.967,-81.356,179.341,16.739,151.697
C02686=1102.138,310.720,-81.325,179.338,16.737,151.698
C02687=1102.133,310.472,-81.294,179.334,16.735,151.698
C02688=1102.127,310.223,-81.262,179.332,16.734,151.698
C02689=1102.121,309.976,-81.232,179.328,16.732,151.698
C02690=1102.116,309.728,-81.200,179.325,16.730,151.699
C02691=1102.109,309.480,-81.169,179.321,16.728,151.699
C02692=1102.104,309.231,-81.138,179.318,16.726,151.699
C02693=1102.098,308.984,-81.107,179.314,16.724,151.700
C02694=1102.093,308.736,-81.076,179.310,16.722,151.700
C02695=1102.087,308.488,-81.046,179.308,16.721,151.700
C02696=1102.081,308.240,-81.014,179.304,16.719,151.700
C02697=1102.076,307.992,-80.983,179.301,16.717,151.701
C02698=1102.070,307.743,-80.952,179.297,16.715,151.701
C02699=1102.064,307.496,-80.921,179.293,16.714,151.701
C02700=1102.059,307.248,-80.890,179.290,16.711,151.701
C02701=1102.053,307.000,-80.859,179.286,16.710,151.702
C02702=1102.047,306.753,-80.828,179.283,16.708,151.702
C02703=1102.042,306.504,-80.797,179.280,16.707,151.702
C02704=1102.036,306.256,-80.767,179.277,16.705,151.702
C02705=1102.031,306.008,-80.736,179.273,16.703,151.703
C02706=1102.025,305.760,-80.705,179.270,16.701,151.703
C02707=1102.018,305.512,-80.674,179.266,16.699,151.703
C02708=1102.013,305.264,-80.643,179.262,16.697,151.704
C02709=1102.007,305.016,-80.613,179.259,16.695,151.704
C02710=1102.002,304.768,-80.582,179.256,16.694,151.704
C02711=1101.996,304.520,-80.551,179.253,16.692,151.704
C02712=1101.991,304.272,-80.520,179.249,16.690,151.705
C02713=1101.985,304.024,-80.490,179.245,16.689,151.705
C02714=1101.979,303.776,-80.459,179.242,16.687,151.705
C02715=1101.971,303.395,-80.411,179.236,16.684,151.706
C02716=1101.963,303.014,-80.364,179.231,16.681,151.706
C02717=1101.954,302.632,-80.317,179.226,16.679,151.707
C02718=1101.945,302.252,-80.271,179.221,16.676,151.707
C02719=1101.939,302.003,-80.240,179.217,16.675,151.707
C02720=1101.934,301.755,-80.209,179.214,16.673,151.708
C02721=1101.928,301.507,-80.178,179.210,16.671,151.708
C02722=1101.923,301.259,-80.148,179.207,16.669,151.708
C02723=1101.917,301.012,-80.118,179.204,16.668,151.708
C02724=1101.912,300.763,-80.087,179.200,16.666,151.709
C02725=1101.906,300.516,-80.056,179.197,16.664,151.709
C02726=1101.900,300.268,-80.026,179.193,16.662,151.709
C02727=1101.895,300.020,-79.995,179.190,16.661,151.710
C02728=1101.890,299.771,-79.966,179.187,16.660,151.710
C02729=1101.884,299.523,-79.935,179.183,16.657,151.710
C02730=1101.879,299.275,-79.904,179.180,16.656,151.711
C02731=1101.873,299.027,-79.874,179.176,16.654,151.711
C02732=1101.867,298.780,-79.844,179.172,16.652,151.711
C02733=1101.861,298.532,-79.813,179.170,16.651,151.712
C02734=1101.856,298.283,-79.783,179.166,16.649,151.712
C02735=1101.851,298.035,-79.753,179.162,16.648,151.712
C02736=1101.845,297.787,-79.722,179.159,16.646,151.713
C02737=1101.839,297.540,-79.692,179.155,16.644,151.713
C02738=1101.833,297.291,-79.662,179.152,16.643,151.713
C02739=1101.828,297.043,-79.632,179.149,16.641,151.713
C02740=1101.822,296.796,-79.602,179.145,16.639,151.714
C02741=1101.817,296.547,-79.571,179.141,16.638,151.714
C02742=1101.811,296.299,-79.541,179.138,16.637,151.715
C02743=1101.805,296.050,-79.510,179.135,16.635,151.715
C02744=1101.799,295.802,-79.481,179.131,16.633,151.715
C02745=1101.793,295.554,-79.450,179.127,16.632,151.716
C02746=1101.788,295.306,-79.420,179.124,16.631,151.716
C02747=1101.782,295.058,-79.390,179.121,16.629,151.716
C02748=1101.776,294.810,-79.360,179.117,16.627,151.717
C02749=1101.771,294.562,-79.330,179.113,16.626,151.717
C02750=1101.765,294.314,-79.300,179.110,16.625,151.717
C02751=1101.760,294.065,-79.270,179.107,16.623,151.718
C02752=1101.754,293.818,-79.240,179.103,16.621,151.718
C02753=1101.749,293.570,-79.211,179.099,16.620,151.718
C02754=1101.743,293.322,-79.180,179.096,16.619,151.719
C02755=1101.737,293.074,-79.151,179.093,16.617,151.719
C02756=1101.732,292.826,-79.120,179.089,16.615,151.720
C02757=1101.726,292.577,-79.091,179.085,16.614,151.720
C02758=1101.720,292.329,-79.060,179.082,16.613,151.720
C02759=1101.715,292.081,-79.031,179.079,16.611,151.721
C02760=1101.708,291.833,-79.001,179.075,16.609,151.721
C02761=1101.703,291.585,-78.971,179.072,16.608,151.721
C02762=1101.697,291.337,-78.942,179.068,16.606,151.722
C02763=1101.691,291.089,-78.911,179.065,16.605,151.722
C02764=1101.686,290.840,-78.882,179.061,16.603,151.722
C02765=1101.680,290.592,-78.852,179.058,16.602,151.723
C02766=1101.675,290.344,-78.822,179.054,16.600,151.723
C02767=1101.667,289.977,-78.778,179.050,16.599,151.724
C02768=1101.658,289.609,-78.734,179.044,16.596,151.724
C02769=1101.650,289.243,-78.690,179.039,16.595,151.725
C02770=1101.641,288.875,-78.647,179.034,16.592,151.725
C02771=1101.635,288.627,-78.617,179.030,16.590,151.726
C02772=1101.629,288.379,-78.587,179.027,16.589,151.726
C02773=1101.624,288.130,-78.557,179.023,16.588,151.727
C02774=1101.618,287.883,-78.528,179.019,16.587,151.727
C02775=1101.613,287.635,-78.499,179.016,16.585,151.727
C02776=1101.607,287.386,-78.469,179.013,16.584,151.728
C02777=1101.602,287.138,-78.439,179.009,16.583,151.728
C02778=1101.595,286.890,-78.410,179.006,16.582,151.729
C02779=1101.590,286.642,-78.380,179.002,16.580,151.729
C02780=1101.584,286.393,-78.350,178.998,16.578,151.729
C02781=1101.578,286.146,-78.322,178.995,16.577,151.730
C02782=1101.573,285.897,-78.292,178.991,16.576,151.730
C02783=1101.567,285.649,-78.262,178.988,16.574,151.731
C02784=1101.561,285.401,-78.233,178.985,16.573,151.731
C02785=1101.556,285.152,-78.204,178.981,16.572,151.731
C02786=1101.551,284.905,-78.174,178.977,16.570,151.732
C02787=1101.545,284.657,-78.145,178.974,16.569,151.732
C02788=1101.539,284.408,-78.116,178.971,16.568,151.733
C02789=1101.534,284.160,-78.086,178.967,16.566,151.733
C02790=1101.527,283.912,-78.057,178.964,16.565,151.733
C02791=1101.522,283.664,-78.028,178.960,16.564,151.734
C02792=1101.517,283.415,-77.998,178.956,16.562,151.734
C02793=1101.511,283.167,-77.969,178.953,16.561,151.734
C02794=1101.505,282.919,-77.940,178.949,16.560,151.735
C02795=1101.499,282.671,-77.911,178.946,16.558,151.735
C02796=1101.494,282.423,-77.881,178.943,16.557,151.736
C02797=1101.488,282.174,-77.852,178.939,16.555,151.736
C02798=1101.482,281.926,-77.823,178.935,16.554,151.737
C02799=1101.478,281.678,-77.794,178.932,16.553,151.737
C02800=1101.471,281.430,-77.765,178.929,16.552,151.737
C02801=1101.466,281.181,-77.735,178.925,16.550,151.738
C02802=1101.460,280.934,-77.707,178.922,16.549,151.738
C02803=1101.455,280.686,-77.677,178.918,16.548,151.739
C02804=1101.449,280.437,-77.649,178.915,16.547,151.739
C02805=1101.443,280.188,-77.619,178.911,16.545,151.739
C02806=1101.438,279.941,-77.590,178.907,16.544,151.740
C02807=1101.432,279.692,-77.561,178.904,16.543,151.740
C02808=1101.426,279.444,-77.532,178.900,16.542,151.741
C02809=1101.421,279.195,-77.503,178.896,16.540,151.741
C02810=1101.415,278.948,-77.474,178.894,16.539,151.742
C02811=1101.409,278.699,-77.446,178.890,16.538,151.742
C02812=1101.403,278.451,-77.416,178.887,16.537,151.742
C02813=1101.398,278.203,-77.388,178.883,16.536,151.743
C02814=1101.393,277.954,-77.359,178.879,16.534,151.743
C02815=1101.386,277.706,-77.330,178.876,16.533,151.744
C02816=1101.381,277.459,-77.301,178.872,16.532,151.744
C02817=1101.376,277.210,-77.272,178.869,16.531,151.745
C02818=1101.369,276.961,-77.243,178.865,16.530,151.745
C02819=1101.362,276.604,-77.202,178.860,16.528,151.746
C02820=1101.353,276.246,-77.161,178.855,16.526,151.746
C02821=1101.345,275.888,-77.118,178.849,16.524,151.747
C02822=1101.337,275.530,-77.077,178.845,16.522,151.748
C02823=1101.331,275.281,-77.048,178.841,16.522,151.748
C02824=1101.326,275.033,-77.020,178.838,16.520,151.749
C02825=1101.320,274.785,-76.991,178.834,16.519,151.749
C02826=1101.315,274.537,-76.963,178.831,16.518,151.749
C02827=1101.309,274.289,-76.934,178.827,16.517,151.750
C02828=1101.303,274.040,-76.905,178.824,16.516,151.750
C02829=1101.298,273.792,-76.877,178.820,16.514,151.751
C02830=1101.292,273.544,-76.848,178.816,16.513,151.751
C02831=1101.286,273.296,-76.820,178.813,16.512,151.752
C02832=1101.280,273.047,-76.791,178.809,16.510,151.752
C02833=1101.275,272.798,-76.762,178.806,16.510,151.753
C02834=1101.270,272.550,-76.734,178.802,16.508,151.753
C02835=1101.263,272.302,-76.705,178.799,16.508,151.754
C02836=1101.258,272.054,-76.677,178.795,16.506,151.754
C02837=1101.252,271.805,-76.648,178.792,16.505,151.754
C02838=1101.246,271.558,-76.620,178.788,16.504,151.755
C02839=1101.241,271.309,-76.591,178.785,16.503,151.755
C02840=1101.236,271.061,-76.563,178.781,16.502,151.756
C02841=1101.230,270.812,-76.535,178.777,16.501,151.756
C02842=1101.224,270.564,-76.506,178.775,16.500,151.757
C02843=1101.218,270.316,-76.478,178.771,16.498,151.757
C02844=1101.212,270.067,-76.449,178.767,16.497,151.758
C02845=1101.207,269.819,-76.421,178.764,16.496,151.758
C02846=1101.201,269.570,-76.393,178.760,16.495,151.759
C02847=1101.196,269.323,-76.364,178.757,16.494,151.759
C02848=1101.190,269.074,-76.336,178.753,16.493,151.760
C02849=1101.184,268.826,-76.308,178.750,16.492,151.760
C02850=1101.178,268.577,-76.280,178.746,16.491,151.760
C02851=1101.173,268.329,-76.252,178.743,16.490,151.761
C02852=1101.167,268.081,-76.223,178.739,16.489,151.762
C02853=1101.162,267.832,-76.195,178.736,16.488,151.762
C02854=1101.155,267.584,-76.166,178.732,16.487,151.762
C02855=1101.150,267.336,-76.138,178.728,16.485,151.763
C02856=1101.144,267.088,-76.110,178.725,16.484,151.763
C02857=1101.139,266.840,-76.082,178.721,16.483,151.764
C02858=1101.133,266.591,-76.054,178.718,16.482,151.764
C02859=1101.127,266.343,-76.026,178.714,16.481,151.765
C02860=1101.122,266.094,-75.998,178.711,16.480,151.765
C02861=1101.116,265.846,-75.970,178.707,16.479,151.766
C02862=1101.111,265.598,-75.942,178.704,16.478,151.766
C02863=1101.105,265.349,-75.913,178.700,16.477,151.767
C02864=1101.100,265.101,-75.885,178.697,16.476,151.767
C02865=1101.094,264.852,-75.858,178.693,16.475,151.768
C02866=1101.089,264.604,-75.830,178.690,16.474,151.768
C02867=1101.083,264.356,-75.802,178.686,16.473,151.769
C02868=1101.077,264.107,-75.773,178.682,16.472,151.769
C02869=1101.071,263.859,-75.746,178.678,16.471,151.770
C02870=1101.065,263.610,-75.718,178.675,16.470,151.770
C02871=1101.057,263.255,-75.678,178.670,16.469,151.771
C02872=1101.049,262.899,-75.638,178.665,16.468,151.772
C02873=1101.040,262.545,-75.598,178.660,16.466,151.772
C02874=1101.032,262.190,-75.558,178.655,16.465,151.773
C02875=1101.027,261.941,-75.531,178.651,16.464,151.774
C02876=1101.021,261.693,-75.503,178.648,16.463,151.774
C02877=1101.015,261.445,-75.475,178.644,16.461,151.775
C02878=1101.009,261.196,-75.447,178.641,16.461,151.775
C02879=1101.004,260.948,-75.420,178.637,16.460,151.776
C02880=1100.998,260.699,-75.392,178.634,16.459,151.776
C02881=1100.992,260.451,-75.364,178.630,16.458,151.777
C02882=1100.987,260.203,-75.336,178.626,16.457,151.777
C02883=1100.981,259.954,-75.309,178.622,16.456,151.778
C02884=1100.975,259.706,-75.281,178.619,16.455,151.778
C02885=1100.970,259.458,-75.253,178.615,16.454,151.779
C02886=1100.964,259.209,-75.226,178.612,16.453,151.779
C02887=1100.958,258.961,-75.198,178.608,16.452,151.780
C02888=1100.952,258.712,-75.172,178.605,16.451,151.780
C02889=1100.947,258.464,-75.143,178.601,16.450,151.781
C02890=1100.941,258.216,-75.115,178.598,16.450,151.781
C02891=1100.935,257.967,-75.089,178.594,16.448,151.782
C02892=1100.929,257.718,-75.060,178.591,16.447,151.782
C02893=1100.924,257.470,-75.033,178.587,16.446,151.783
C02894=1100.918,257.222,-75.006,178.584,16.446,151.783
C02895=1100.913,256.973,-74.978,178.580,16.445,151.784
C02896=1100.907,256.725,-74.951,178.576,16.444,151.784
C02897=1100.902,256.476,-74.924,178.572,16.443,151.785
C02898=1100.896,256.228,-74.896,178.569,16.442,151.785
C02899=1100.890,255.979,-74.869,178.565,16.441,151.786
C02900=1100.885,255.731,-74.841,178.562,16.440,151.786
C02901=1100.879,255.483,-74.814,178.559,16.439,151.787
C02902=1100.873,255.234,-74.786,178.555,16.438,151.787
C02903=1100.867,254.986,-74.759,178.552,16.438,151.788
C02904=1100.862,254.737,-74.732,178.548,16.436,151.788
C02905=1100.856,254.489,-74.704,178.545,16.436,151.789
C02906=1100.851,254.241,-74.677,178.541,16.435,151.790
C02907=1100.845,253.991,-74.650,178.537,16.434,151.790
C02908=1100.839,253.743,-74.622,178.534,16.432,151.790
C02909=1100.833,253.495,-74.596,178.530,16.432,151.791
C02910=1100.828,253.246,-74.568,178.526,16.431,151.792
C02911=1100.822,252.999,-74.541,178.523,16.430,151.792
C02912=1100.817,252.749,-74.513,178.520,16.430,151.793
C02913=1100.811,252.501,-74.487,178.516,16.428,151.793
C02914=1100.806,252.252,-74.459,178.513,16.428,151.794
C02915=1100.800,252.004,-74.432,178.509,16.427,151.794
C02916=1100.795,251.756,-74.405,178.506,16.426,151.795
C02917=1100.789,251.507,-74.378,178.502,16.424,151.795
C02918=1100.783,251.258,-74.351,178.499,16.424,151.796
C02919=1100.777,251.010,-74.323,178.495,16.423,151.796
C02920=1100.772,250.762,-74.296,178.491,16.422,151.797
C02921=1100.766,250.513,-74.269,178.488,16.422,151.797
C02922=1100.761,250.265,-74.242,178.484,16.420,151.798
C02923=1100.753,249.907,-74.203,178.479,16.419,151.799
C02924=1100.745,249.548,-74.165,178.474,16.418,151.799
C02925=1100.737,249.191,-74.126,178.469,16.416,151.800
C02926=1100.730,248.833,-74.086,178.464,16.415,151.801
C02927=1100.723,248.584,-74.059,178.461,16.414,151.801
C02928=1100.717,248.336,-74.033,178.457,16.413,151.802
C02929=1100.712,248.087,-74.005,178.453,16.413,151.802
C02930=1100.707,247.839,-73.979,178.450,16.412,151.803
C02931=1100.702,247.590,-73.952,178.446,16.411,151.803
C02932=1100.696,247.342,-73.925,178.443,16.410,151.804
C02933=1100.690,247.093,-73.898,178.439,16.409,151.804
C02934=1100.684,246.845,-73.872,178.436,16.408,151.805
C02935=1100.679,246.596,-73.844,178.433,16.408,151.806
C02936=1100.673,246.348,-73.818,178.429,16.407,151.806
C02937=1100.668,246.100,-73.791,178.425,16.406,151.807
C02938=1100.662,245.851,-73.764,178.421,16.405,151.807
C02939=1100.656,245.602,-73.739,178.418,16.404,151.808
C02940=1100.651,245.354,-73.711,178.415,16.404,151.808
C02941=1100.646,245.105,-73.685,178.411,16.403,151.809
C02942=1100.639,244.856,-73.658,178.408,16.402,151.809
C02943=1100.633,244.608,-73.631,178.404,16.401,151.810
C02944=1100.628,244.359,-73.604,178.400,16.400,151.810
C02945=1100.623,244.111,-73.577,178.397,16.400,151.811
C02946=1100.617,243.862,-73.551,178.393,16.399,151.812
C02947=1100.611,243.613,-73.524,178.390,16.398,151.812
C02948=1100.606,243.365,-73.498,178.386,16.397,151.813
C02949=1100.600,243.117,-73.471,178.383,16.396,151.813
C02950=1100.594,242.868,-73.445,178.379,16.396,151.814
C02951=1100.589,242.619,-73.419,178.375,16.395,151.814
C02952=1100.583,242.371,-73.392,178.372,16.394,151.815
C02953=1100.578,242.122,-73.365,178.369,16.393,151.815
C02954=1100.572,241.874,-73.338,178.365,16.392,151.816
C02955=1100.567,241.625,-73.312,178.362,16.392,151.816
C02956=1100.561,241.377,-73.285,178.357,16.391,151.817
C02957=1100.555,241.128,-73.259,178.354,16.390,151.818
C02958=1100.550,240.879,-73.233,178.351,16.390,151.818
C02959=1100.544,240.631,-73.206,178.347,16.389,151.819
C02960=1100.538,240.383,-73.180,178.344,16.388,151.819
C02961=1100.533,240.134,-73.154,178.341,16.388,151.820
C02962=1100.527,239.885,-73.127,178.337,16.386,151.820
C02963=1100.521,239.636,-73.101,178.333,16.386,151.821
C02964=1100.515,239.388,-73.075,178.329,16.385,151.821
C02965=1100.509,239.140,-73.048,178.326,16.384,151.822
C02966=1100.504,238.892,-73.023,178.323,16.384,151.823
C02967=1100.498,238.643,-72.996,178.319,16.383,151.823
C02968=1100.493,238.394,-72.970,178.315,16.382,151.824
C02969=1100.487,238.146,-72.944,178.312,16.382,151.824
C02970=1100.482,237.897,-72.918,178.308,16.381,151.825
C02971=1100.476,237.649,-72.891,178.305,16.380,151.825
C02972=1100.470,237.400,-72.865,178.302,16.380,151.826
C02973=1100.465,237.151,-72.838,178.298,16.378,151.826
C02974=1100.459,236.902,-72.812,178.294,16.378,151.827
C02975=1100.451,236.538,-72.774,178.289,16.377,151.828
C02976=1100.442,236.173,-72.736,178.284,16.376,151.829
C02977=1100.434,235.808,-72.698,178.279,16.375,151.830
C02978=1100.426,235.443,-72.660,178.273,16.373,151.830
C02979=1100.420,235.195,-72.633,178.270,16.373,151.831
C02980=1100.415,234.946,-72.607,178.267,16.373,151.832
C02981=1100.409,234.697,-72.581,178.263,16.371,151.832
C02982=1100.404,234.449,-72.555,178.259,16.371,151.833
C02983=1100.397,234.200,-72.529,178.256,16.370,151.833
C02984=1100.393,233.952,-72.504,178.252,16.369,151.834
C02985=1100.387,233.704,-72.477,178.249,16.369,151.834
C02986=1100.381,233.455,-72.451,178.246,16.368,151.835
C02987=1100.375,233.206,-72.426,178.241,16.367,151.835
C02988=1100.369,232.957,-72.399,178.238,16.367,151.836
C02989=1100.365,232.709,-72.374,178.235,16.366,151.837
C02990=1100.359,232.460,-72.348,178.231,16.365,151.837
C02991=1100.353,232.212,-72.322,178.228,16.365,151.838
C02992=1100.347,231.963,-72.296,178.225,16.364,151.838
C02993=1100.342,231.714,-72.270,178.221,16.364,151.839
C02994=1100.337,231.466,-72.244,178.217,16.363,151.839
C02995=1100.331,231.217,-72.219,178.214,16.362,151.840
C02996=1100.325,230.968,-72.193,178.211,16.362,151.841
C02997=1100.320,230.719,-72.167,178.207,16.361,151.841
C02998=1100.313,230.471,-72.142,178.203,16.360,151.842
C02999=1100.308,230.223,-72.115,178.200,16.359,151.842
C03000=1100.303,229.974,-72.089,178.196,16.359,151.843
C03001=1100.297,229.725,-72.064,178.193,16.358,151.843
C03002=1100.291,229.476,-72.038,178.189,16.358,151.844
C03003=1100.285,229.228,-72.013,178.186,16.357,151.845
C03004=1100.280,228.979,-71.987,178.182,16.356,151.845
C03005=1100.274,228.731,-71.962,178.179,16.356,151.846
C03006=1100.268,228.482,-71.936,178.175,16.355,151.846
C03007=1100.262,228.233,-71.911,178.171,16.354,151.847
C03008=1100.257,227.985,-71.885,178.168,16.354,151.847
C03009=1100.251,227.736,-71.860,178.165,16.353,151.848
C03010=1100.246,227.487,-71.834,178.161,16.353,151.849
C03011=1100.241,227.239,-71.808,178.157,16.352,151.849
C03012=1100.235,226.990,-71.783,178.154,16.351,151.850
C03013=1100.229,226.741,-71.757,178.151,16.351,151.850
C03014=1100.223,226.493,-71.732,178.147,16.350,151.851
C03015=1100.218,226.244,-71.706,178.143,16.350,151.852
C03016=1100.212,225.996,-71.681,178.140,16.349,151.852
C03017=1100.206,225.747,-71.655,178.137,16.348,151.853
C03018=1100.201,225.499,-71.630,178.133,16.347,151.853
C03019=1100.195,225.249,-71.605,178.130,16.347,151.854
C03020=1100.189,225.000,-71.579,178.126,16.347,151.854
C03021=1100.184,224.752,-71.554,178.122,16.346,151.855
C03022=1100.178,224.503,-71.528,178.119,16.345,151.856
C03023=1100.172,224.255,-71.503,178.116,16.344,151.856
C03024=1100.167,224.007,-71.478,178.112,16.344,151.857
C03025=1100.161,223.757,-71.453,178.108,16.343,151.857
C03026=1100.156,223.508,-71.427,178.105,16.343,151.858
C03027=1100.147,223.136,-71.389,178.099,16.342,151.859
C03028=1100.139,222.762,-71.351,178.094,16.341,151.860
C03029=1100.130,222.390,-71.314,178.089,16.340,151.861
C03030=1100.122,222.016,-71.276,178.084,16.339,151.861
C03031=1100.116,221.767,-71.250,178.080,16.338,151.862
C03032=1100.111,221.518,-71.226,178.077,16.338,151.863
C03033=1100.105,221.270,-71.200,178.074,16.338,151.863
C03034=1100.099,221.021,-71.174,178.070,16.337,151.864
C03035=1100.094,220.772,-71.150,178.066,16.336,151.864
C03036=1100.088,220.523,-71.125,178.063,16.336,151.865
C03037=1100.082,220.275,-71.100,178.059,16.335,151.866
C03038=1100.077,220.026,-71.075,178.056,16.335,151.866
C03039=1100.071,219.777,-71.049,178.052,16.334,151.867
C03040=1100.065,219.529,-71.024,178.049,16.334,151.867
C03041=1100.059,219.280,-71.000,178.045,16.333,151.868
C03042=1100.054,219.032,-70.975,178.042,16.333,151.868
C03043=1100.049,218.782,-70.950,178.039,16.332,151.869
C03044=1100.043,218.534,-70.925,178.035,16.331,151.870
C03045=1100.037,218.285,-70.900,178.031,16.331,151.870
C03046=1100.031,218.036,-70.875,178.028,16.330,151.871
C03047=1100.026,217.788,-70.850,178.025,16.330,151.872
C03048=1100.020,217.539,-70.824,178.021,16.329,151.872
C03049=1100.015,217.290,-70.800,178.017,16.329,151.873
C03050=1100.009,217.041,-70.775,178.014,16.328,151.873
C03051=1100.003,216.793,-70.751,178.011,16.328,151.874
C03052=1099.997,216.544,-70.725,178.007,16.327,151.874
C03053=1099.992,216.296,-70.701,178.003,16.326,151.875
C03054=1099.986,216.047,-70.675,178.000,16.326,151.876
C03055=1099.981,215.798,-70.651,177.997,16.325,151.876
C03056=1099.975,215.549,-70.626,177.993,16.325,151.877
C03057=1099.970,215.301,-70.601,177.989,16.324,151.877
C03058=1099.964,215.052,-70.577,177.986,16.323,151.878
C03059=1099.958,214.803,-70.552,177.983,16.323,151.879
C03060=1099.953,214.555,-70.527,177.979,16.323,151.879
C03061=1099.948,214.305,-70.502,177.976,16.322,151.880
C03062=1099.942,214.057,-70.478,177.972,16.321,151.880
C03063=1099.936,213.808,-70.453,177.969,16.321,151.881
C03064=1099.931,213.559,-70.428,177.965,16.321,151.882
C03065=1099.925,213.310,-70.404,177.962,16.320,151.882
C03066=1099.919,213.062,-70.379,177.959,16.320,151.883
C03067=1099.914,212.814,-70.354,177.955,16.318,151.883
C03068=1099.908,212.564,-70.330,177.951,16.318,151.884
C03069=1099.903,212.316,-70.306,177.948,16.318,151.885
C03070=1099.897,212.067,-70.280,177.945,16.317,151.885
C03071=1099.891,211.819,-70.256,177.941,16.317,151.886
C03072=1099.885,211.569,-70.231,177.937,16.316,151.886
C03073=1099.880,211.321,-70.207,177.934,16.316,151.887
C03074=1099.875,211.072,-70.183,177.931,16.315,151.887
C03075=1099.869,210.823,-70.157,177.927,16.315,151.888
C03076=1099.863,210.575,-70.133,177.924,16.315,151.889
C03077=1099.857,210.326,-70.109,177.921,16.314,151.889
C03078=1099.851,210.077,-70.085,177.916,16.313,151.890
C03079=1099.843,209.708,-70.049,177.912,16.313,151.891
C03080=1099.835,209.338,-70.013,177.907,16.312,151.892
C03081=1099.827,208.968,-69.976,177.901,16.311,151.893
C03082=1099.818,208.600,-69.940,177.896,16.310,151.893
C03083=1099.795,207.591,-69.842,177.856,16.298,151.899
C03084=1099.790,207.343,-69.818,177.853,16.298,151.900
C03085=1099.784,207.094,-69.794,177.849,16.299,151.901
C03086=1099.778,206.845,-69.770,177.845,16.299,151.902
C03087=1099.773,206.596,-69.745,177.841,16.300,151.902
C03088=1099.767,206.348,-69.722,177.837,16.300,151.903
C03089=1099.761,206.099,-69.697,177.834,16.301,151.904
C03090=1099.756,205.850,-69.673,177.831,16.301,151.905
C03091=1099.750,205.601,-69.650,177.827,16.301,151.906
C03092=1099.745,205.353,-69.626,177.823,16.302,151.907
C03093=1099.739,205.104,-69.601,177.819,16.302,151.907
C03094=1099.733,204.855,-69.577,177.816,16.302,151.908
C03095=1099.728,204.606,-69.554,177.812,16.302,151.909
C03096=1099.722,204.357,-69.530,177.808,16.302,151.910
C03097=1099.716,204.109,-69.506,177.805,16.303,151.911
C03098=1099.710,203.860,-69.481,177.801,16.304,151.911
C03099=1099.705,203.611,-69.458,177.797,16.304,151.912
C03100=1099.699,203.362,-69.434,177.794,16.304,151.913
C03101=1099.694,203.114,-69.410,177.790,16.304,151.914
C03102=1099.689,202.865,-69.386,177.786,16.305,151.915
C03103=1099.683,202.616,-69.362,177.783,16.305,151.916
C03104=1099.676,202.367,-69.339,177.780,16.306,151.916
C03105=1099.671,202.119,-69.314,177.776,16.306,151.917
C03106=1099.665,201.870,-69.291,177.772,16.307,151.918
C03107=1099.660,201.621,-69.267,177.768,16.307,151.919
C03108=1099.654,201.372,-69.243,177.765,16.307,151.920
C03109=1099.649,201.123,-69.220,177.761,16.307,151.921
C03110=1099.642,200.875,-69.196,177.757,16.308,151.921
C03111=1099.637,200.625,-69.172,177.754,16.308,151.922
C03112=1099.631,200.377,-69.148,177.750,16.309,151.923
C03113=1099.625,200.128,-69.125,177.746,16.309,151.924
C03114=1099.620,199.879,-69.101,177.743,16.310,151.925
C03115=1099.614,199.631,-69.077,177.739,16.310,151.926
C03116=1099.608,199.381,-69.054,177.735,16.310,151.926
C03117=1099.602,199.133,-69.030,177.731,16.310,151.927
C03118=1099.596,198.884,-69.007,177.729,16.311,151.928
C03119=1099.591,198.635,-68.983,177.725,16.311,151.929
C03120=1099.585,198.386,-68.960,177.721,16.312,151.930
C03121=1099.580,198.138,-68.935,177.717,16.312,151.930
C03122=1099.574,197.888,-68.912,177.714,16.312,151.931
C03123=1099.568,197.640,-68.888,177.710,16.312,151.932
C03124=1099.563,197.391,-68.865,177.707,16.313,151.933
C03125=1099.557,197.142,-68.841,177.703,16.313,151.934
C03126=1099.551,196.893,-68.818,177.700,16.313,151.934
C03127=1099.546,196.644,-68.795,177.696,16.314,151.935
C03128=1099.540,196.396,-68.771,177.692,16.314,151.936
C03129=1099.534,196.147,-68.748,177.688,16.314,151.937
C03130=1099.529,195.899,-68.724,177.685,16.315,151.938
C03131=1099.523,195.649,-68.701,177.682,16.315,151.938
C03132=1099.517,195.400,-68.678,177.678,16.316,151.939
C03133=1099.512,195.151,-68.653,177.674,16.316,151.940
C03134=1099.506,194.903,-68.630,177.671,16.316,151.941
C03135=1099.500,194.654,-68.608,177.667,16.316,151.942
C03136=1099.495,194.405,-68.583,177.663,16.316,151.943
C03137=1099.489,194.156,-68.560,177.660,16.317,151.943
C03138=1099.483,193.907,-68.537,177.657,16.317,151.944
C03139=1099.478,193.658,-68.514,177.653,16.318,151.945
C03140=1099.472,193.410,-68.490,177.649,16.318,151.946
C03141=1099.467,193.161,-68.467,177.645,16.318,151.947
C03142=1099.461,192.912,-68.444,177.642,16.318,151.947
C03143=1099.456,192.663,-68.421,177.639,16.319,151.948
C03144=1099.449,192.389,-68.395,177.635,16.319,151.949
C03145=1099.443,192.117,-68.370,177.631,16.319,151.950
C03146=1099.437,191.843,-68.345,177.627,16.319,151.951
C03147=1099.430,191.570,-68.319,177.623,16.320,151.952
C03148=1099.425,191.320,-68.295,177.619,16.320,151.952
C03149=1099.419,191.071,-68.272,177.616,16.321,151.953
C03150=1099.414,190.822,-68.249,177.613,16.321,151.954
C03151=1099.408,190.575,-68.226,177.609,16.321,151.955
C03152=1099.403,190.326,-68.203,177.605,16.321,151.955
C03153=1099.398,190.077,-68.179,177.601,16.322,151.956
C03154=1099.392,189.828,-68.156,177.598,16.322,151.957
C03155=1099.386,189.579,-68.133,177.595,16.322,151.958
C03156=1099.380,189.330,-68.110,177.591,16.323,151.959
C03157=1099.375,189.081,-68.088,177.588,16.323,151.959
C03158=1099.370,188.832,-68.064,177.584,16.323,151.960
C03159=1099.364,188.583,-68.041,177.580,16.323,151.961
C03160=1099.358,188.334,-68.018,177.577,16.323,151.962
C03161=1099.352,188.085,-67.995,177.574,16.324,151.963
C03162=1099.347,187.836,-67.972,177.570,16.324,151.963
C03163=1099.341,187.588,-67.949,177.567,16.324,151.964
C03164=1099.337,187.339,-67.926,177.563,16.324,151.965
C03165=1099.331,187.090,-67.903,177.559,16.324,151.966
C03166=1099.325,186.841,-67.880,177.557,16.325,151.966
C03167=1099.319,186.592,-67.857,177.553,16.325,151.967
C03168=1099.314,186.343,-67.834,177.549,16.325,151.968
C03169=1099.308,186.095,-67.811,177.546,16.325,151.969
C03170=1099.302,185.846,-67.788,177.542,16.325,151.969
C03171=1099.297,185.596,-67.765,177.539,16.325,151.970
C03172=1099.292,185.348,-67.743,177.536,16.326,151.971
C03173=1099.287,185.099,-67.720,177.532,16.326,151.972
C03174=1099.281,184.850,-67.697,177.528,16.326,151.972
C03175=1099.274,184.601,-67.675,177.525,16.327,151.973
C03176=1099.269,184.352,-67.652,177.521,16.327,151.974
C03177=1099.263,184.103,-67.629,177.518,16.328,151.975
C03178=1099.257,183.855,-67.606,177.514,16.328,151.975
C03179=1099.252,183.606,-67.583,177.511,16.328,151.976
C03180=1099.246,183.356,-67.561,177.507,16.328,151.977
C03181=1099.240,183.108,-67.538,177.504,16.329,151.978
C03182=1099.234,182.859,-67.515,177.500,16.329,151.979
C03183=1099.228,182.610,-67.493,177.497,16.329,151.979
C03184=1099.222,182.361,-67.470,177.493,16.329,151.980
C03185=1099.218,182.112,-67.448,177.489,16.330,151.981
C03186=1099.211,181.863,-67.425,177.487,16.330,151.982
C03187=1099.205,181.615,-67.402,177.483,16.330,151.982
C03188=1099.200,181.366,-67.379,177.479,16.331,151.983
C03189=1099.194,181.116,-67.357,177.476,16.331,151.984
C03190=1099.188,180.868,-67.335,177.472,16.331,151.985
C03191=1099.182,180.619,-67.312,177.469,16.332,151.986
C03192=1099.177,180.369,-67.290,177.466,16.332,151.986
C03193=1099.171,180.121,-67.267,177.462,16.332,151.987
C03194=1099.166,179.872,-67.244,177.459,16.332,151.988
C03195=1099.160,179.623,-67.223,177.455,16.333,151.989
C03196=1099.154,179.374,-67.200,177.452,16.333,151.989
C03197=1099.148,179.125,-67.177,177.448,16.333,151.990
C03198=1099.142,178.876,-67.155,177.445,16.333,151.991
C03199=1099.137,178.628,-67.132,177.441,16.333,151.992
C03200=1099.131,178.378,-67.110,177.438,16.334,151.992
C03201=1099.126,178.129,-67.087,177.435,16.334,151.993
C03202=1099.119,177.881,-67.065,177.431,16.334,151.994
C03203=1099.114,177.631,-67.043,177.427,16.334,151.995
C03204=1099.109,177.383,-67.020,177.425,16.335,151.995
C03205=1099.103,177.134,-66.998,177.421,16.335,151.996
C03206=1099.097,176.885,-66.976,177.417,16.335,151.997
C03207=1099.091,176.635,-66.953,177.414,16.335,151.998
C03208=1099.085,176.362,-66.929,177.410,16.335,151.998
C03209=1099.079,176.088,-66.904,177.407,16.335,151.999
C03210=1099.073,175.815,-66.880,177.403,16.336,152.000
C03211=1099.066,175.541,-66.856,177.399,16.336,152.001
C03212=1099.061,175.291,-66.833,177.395,16.336,152.002
C03213=1099.055,175.043,-66.811,177.393,16.337,152.002
C03214=1099.049,174.794,-66.789,177.389,16.337,152.003
C03215=1099.044,174.545,-66.766,177.385,16.337,152.004
C03216=1099.039,174.296,-66.744,177.382,16.337,152.005
C03217=1099.032,174.048,-66.722,177.378,16.337,152.005
C03218=1099.027,173.798,-66.700,177.376,16.337,152.006
C03219=1099.021,173.550,-66.678,177.372,16.337,152.007
C03220=1099.016,173.301,-66.655,177.368,16.337,152.007
C03221=1099.010,173.051,-66.633,177.365,16.337,152.008
C03222=1099.004,172.802,-66.612,177.362,16.338,152.009
C03223=1098.999,172.554,-66.589,177.359,16.338,152.010
C03224=1098.993,172.304,-66.567,177.355,16.338,152.010
C03225=1098.987,172.055,-66.545,177.351,16.338,152.011
C03226=1098.982,171.807,-66.523,177.349,16.339,152.012
C03227=1098.976,171.558,-66.501,177.345,16.339,152.012
C03228=1098.971,171.309,-66.479,177.342,16.339,152.013
C03229=1098.965,171.060,-66.457,177.338,16.339,152.014
C03230=1098.959,170.811,-66.434,177.335,16.339,152.015
C03231=1098.954,170.562,-66.413,177.332,16.339,152.015
C03232=1098.948,170.313,-66.391,177.328,16.339,152.016
C03233=1098.943,170.063,-66.369,177.325,16.339,152.017
C03234=1098.937,169.815,-66.347,177.322,16.340,152.017
C03235=1098.932,169.566,-66.325,177.318,16.340,152.018
C03236=1098.926,169.317,-66.303,177.315,16.340,152.019
C03237=1098.921,169.068,-66.281,177.311,16.340,152.020
C03238=1098.914,168.819,-66.259,177.309,16.340,152.020
C03239=1098.910,168.570,-66.238,177.305,16.340,152.021
C03240=1098.903,168.321,-66.215,177.302,16.340,152.022
C03241=1098.898,168.072,-66.193,177.298,16.340,152.022
C03242=1098.892,167.823,-66.172,177.295,16.341,152.023
C03243=1098.887,167.574,-66.150,177.292,16.341,152.024
C03244=1098.881,167.325,-66.128,177.288,16.341,152.025
C03245=1098.876,167.076,-66.106,177.285,16.341,152.025
C03246=1098.870,166.827,-66.085,177.282,16.341,152.026
C03247=1098.865,166.578,-66.063,177.279,16.341,152.027
C03248=1098.859,166.329,-66.041,177.275,16.341,152.027
C03249=1098.854,166.080,-66.019,177.272,16.341,152.028
C03250=1098.848,165.831,-65.998,177.269,16.342,152.029
C03251=1098.843,165.582,-65.976,177.266,16.341,152.029
C03252=1098.837,165.333,-65.954,177.262,16.341,152.030
C03253=1098.832,165.084,-65.932,177.259,16.341,152.031
C03254=1098.826,164.835,-65.911,177.256,16.342,152.031
C03255=1098.821,164.586,-65.889,177.252,16.341,152.032
C03256=1098.815,164.337,-65.867,177.249,16.341,152.033
C03257=1098.810,164.088,-65.845,177.245,16.341,152.033
C03258=1098.804,163.839,-65.824,177.243,16.342,152.034
C03259=1098.799,163.591,-65.802,177.239,16.342,152.035
C03260=1098.793,163.341,-65.780,177.236,16.342,152.035
C03261=1098.788,163.093,-65.759,177.232,16.342,152.036
C03262=1098.782,162.843,-65.737,177.230,16.342,152.037
C03263=1098.777,162.595,-65.715,177.226,16.342,152.037
C03264=1098.771,162.346,-65.694,177.223,16.342,152.038
C03265=1098.766,162.096,-65.673,177.219,16.341,152.039
C03266=1098.760,161.847,-65.651,177.217,16.342,152.039
C03267=1098.755,161.598,-65.629,177.213,16.342,152.040
C03268=1098.749,161.349,-65.608,177.210,16.342,152.041
C03269=1098.743,161.100,-65.586,177.206,16.342,152.041
C03270=1098.738,160.852,-65.565,177.204,16.342,152.042
C03271=1098.732,160.602,-65.544,177.200,16.342,152.043
C03272=1098.726,160.328,-65.520,177.196,16.342,152.044
C03273=1098.719,160.054,-65.497,177.193,16.342,152.044
C03274=1098.713,159.780,-65.473,177.189,16.342,152.045
C03275=1098.707,159.507,-65.449,177.186,16.342,152.046
C03276=1098.701,159.257,-65.428,177.182,16.342,152.047
C03277=1098.696,159.008,-65.407,177.180,16.343,152.047
C03278=1098.690,158.759,-65.385,177.176,16.343,152.048
C03279=1098.685,158.510,-65.364,177.173,16.343,152.049
C03280=1098.679,158.260,-65.343,177.169,16.342,152.049
C03281=1098.674,158.012,-65.322,177.167,16.343,152.050
C03282=1098.667,157.763,-65.300,177.163,16.343,152.051
C03283=1098.662,157.513,-65.279,177.160,16.342,152.051
C03284=1098.657,157.265,-65.258,177.157,16.343,152.052
C03285=1098.650,157.016,-65.236,177.154,16.343,152.053
C03286=1098.646,156.766,-65.215,177.150,16.343,152.053
C03287=1098.640,156.517,-65.194,177.147,16.343,152.054
C03288=1098.634,156.269,-65.172,177.144,16.343,152.054
C03289=1098.629,156.020,-65.152,177.141,16.343,152.055
C03290=1098.623,155.770,-65.130,177.137,16.343,152.056
C03291=1098.617,155.521,-65.110,177.135,16.343,152.056
C03292=1098.612,155.273,-65.088,177.131,16.343,152.057
C03293=1098.606,155.023,-65.067,177.128,16.343,152.058
C03294=1098.600,154.774,-65.046,177.124,16.343,152.058
C03295=1098.594,154.525,-65.025,177.122,16.343,152.059
C03296=1098.589,154.276,-65.004,177.118,16.343,152.060
C03297=1098.583,154.028,-64.983,177.115,16.343,152.060
C03298=1098.578,153.778,-64.962,177.112,16.343,152.061
C03299=1098.572,153.529,-64.941,177.109,16.343,152.062
C03300=1098.567,153.280,-64.920,177.105,16.343,152.062
C03301=1098.561,153.031,-64.898,177.103,16.343,152.063
C03302=1098.555,152.782,-64.878,177.099,16.343,152.064
C03303=1098.550,152.533,-64.857,177.096,16.343,152.064
C03304=1098.544,152.283,-64.836,177.093,16.343,152.065
C03305=1098.538,152.035,-64.814,177.090,16.343,152.066
C03306=1098.533,151.786,-64.794,177.087,16.343,152.066
C03307=1098.527,151.537,-64.772,177.083,16.343,152.067
C03308=1098.522,151.287,-64.752,177.081,16.343,152.067
C03309=1098.516,151.038,-64.731,177.077,16.343,152.068
C03310=1098.510,150.789,-64.709,177.074,16.343,152.069
C03311=1098.504,150.540,-64.689,177.071,16.343,152.069
C03312=1098.499,150.292,-64.668,177.068,16.343,152.070
C03313=1098.494,150.043,-64.648,177.064,16.343,152.071
C03314=1098.488,149.793,-64.627,177.061,16.343,152.071
C03315=1098.482,149.544,-64.605,177.058,16.343,152.072
C03316=1098.477,149.295,-64.585,177.055,16.343,152.073
C03317=1098.471,149.045,-64.564,177.052,16.342,152.073
C03318=1098.465,148.797,-64.543,177.049,16.343,152.074
C03319=1098.459,148.548,-64.523,177.046,16.343,152.074
C03320=1098.454,148.299,-64.502,177.042,16.342,152.075
C03321=1098.448,148.049,-64.481,177.040,16.343,152.076
C03322=1098.443,147.801,-64.460,177.036,16.342,152.076
C03323=1098.438,147.552,-64.439,177.033,16.342,152.077
C03324=1098.432,147.303,-64.419,177.030,16.343,152.078
C03325=1098.425,147.053,-64.398,177.027,16.342,152.078
C03326=1098.420,146.804,-64.377,177.023,16.342,152.079
C03327=1098.415,146.555,-64.357,177.021,16.342,152.079
C03328=1098.409,146.306,-64.337,177.017,16.342,152.080
C03329=1098.403,146.057,-64.316,177.014,16.342,152.081
C03330=1098.397,145.808,-64.295,177.011,16.342,152.081
C03331=1098.392,145.559,-64.274,177.008,16.342,152.082
C03332=1098.386,145.310,-64.254,177.005,16.342,152.083
C03333=1098.380,145.060,-64.233,177.002,16.341,152.083
C03334=1098.375,144.811,-64.213,176.999,16.342,152.084
C03335=1098.369,144.562,-64.193,176.996,16.342,152.085
C03336=1098.363,144.288,-64.170,176.992,16.342,152.085
C03337=1098.356,144.013,-64.147,176.989,16.341,152.086
C03338=1098.351,143.739,-64.124,176.985,16.341,152.087
C03339=1098.344,143.465,-64.102,176.982,16.341,152.087
C03340=1098.339,143.216,-64.081,176.979,16.342,152.088
C03341=1098.334,142.967,-64.061,176.976,16.341,152.088
C03342=1098.327,142.717,-64.041,176.973,16.341,152.089
C03343=1098.322,142.468,-64.020,176.970,16.341,152.090
C03344=1098.317,142.219,-63.999,176.967,16.341,152.090
C03345=1098.311,141.970,-63.979,176.963,16.341,152.091
C03346=1098.305,141.722,-63.958,176.961,16.341,152.091
C03347=1098.300,141.473,-63.938,176.958,16.340,152.092
C03348=1098.294,141.224,-63.918,176.954,16.340,152.093
C03349=1098.288,140.974,-63.897,176.952,16.341,152.093
C03350=1098.283,140.724,-63.877,176.948,16.340,152.094
C03351=1098.277,140.476,-63.857,176.945,16.340,152.094
C03352=1098.272,140.226,-63.836,176.943,16.340,152.095
C03353=1098.266,139.978,-63.816,176.939,16.340,152.096
C03354=1098.261,139.729,-63.796,176.936,16.339,152.096
C03355=1098.255,139.480,-63.776,176.933,16.340,152.097
C03356=1098.249,139.231,-63.755,176.930,16.339,152.097
C03357=1098.243,138.981,-63.734,176.927,16.339,152.098
C03358=1098.237,138.732,-63.715,176.924,16.339,152.099
C03359=1098.232,138.483,-63.694,176.921,16.339,152.099
C03360=1098.226,138.234,-63.674,176.918,16.338,152.100
C03361=1098.221,137.985,-63.653,176.915,16.339,152.100
C03362=1098.215,137.736,-63.634,176.912,16.339,152.101
C03363=1098.210,137.486,-63.614,176.909,16.338,152.102
C03364=1098.204,137.238,-63.594,176.906,16.339,152.102
C03365=1098.199,136.988,-63.573,176.903,16.338,152.103
C03366=1098.193,136.740,-63.553,176.900,16.338,152.103
C03367=1098.186,136.490,-63.533,176.897,16.338,152.104
C03368=1098.181,136.240,-63.513,176.894,16.338,152.104
C03369=1098.175,135.991,-63.493,176.891,16.337,152.105
C03370=1098.170,135.742,-63.473,176.888,16.337,152.106
C03371=1098.164,135.494,-63.453,176.885,16.337,152.106
C03372=1098.159,135.244,-63.432,176.882,16.337,152.107
C03373=1098.153,134.995,-63.413,176.879,16.337,152.107
C03374=1098.147,134.746,-63.393,176.876,16.337,152.108
C03375=1098.142,134.497,-63.372,176.873,16.337,152.109
C03376=1098.136,134.248,-63.352,176.870,16.337,152.109
C03377=1098.131,133.999,-63.332,176.867,16.336,152.110
C03378=1098.125,133.750,-63.313,176.864,16.336,152.110
C03379=1098.120,133.501,-63.292,176.861,16.336,152.111
C03380=1098.114,133.251,-63.273,176.858,16.336,152.111
C03381=1098.108,133.002,-63.253,176.855,16.335,152.112
C03382=1098.103,132.753,-63.232,176.852,16.335,152.112
C03383=1098.097,132.504,-63.213,176.849,16.335,152.113
C03384=1098.091,132.255,-63.193,176.846,16.335,152.113
C03385=1098.086,132.006,-63.172,176.843,16.334,152.114
C03386=1098.080,131.756,-63.153,176.840,16.334,152.115
C03387=1098.074,131.508,-63.133,176.837,16.334,152.115
C03388=1098.068,131.258,-63.114,176.834,16.334,152.116
C03389=1098.063,131.009,-63.093,176.832,16.334,152.116
C03390=1098.057,130.760,-63.073,176.828,16.334,152.117
C03391=1098.051,130.511,-63.054,176.825,16.333,152.117
C03392=1098.045,130.262,-63.034,176.823,16.333,152.118
C03393=1098.040,130.013,-63.015,176.819,16.333,152.119
C03394=1098.034,129.763,-62.994,176.816,16.333,152.119
C03395=1098.029,129.514,-62.975,176.814,16.333,152.120
C03396=1098.023,129.265,-62.955,176.810,16.332,152.120
C03397=1098.017,129.016,-62.936,176.808,16.333,152.121
C03398=1098.011,128.767,-62.916,176.805,16.332,152.121
C03399=1098.005,128.517,-62.897,176.801,16.332,152.122
C03400=1097.999,128.244,-62.875,176.798,16.331,152.123
C03401=1097.993,127.969,-62.853,176.795,16.331,152.123
C03402=1097.987,127.694,-62.831,176.792,16.331,152.124
C03403=1097.981,127.420,-62.810,176.789,16.331,152.124
C03404=1097.975,127.171,-62.790,176.786,16.330,152.125
C03405=1097.969,126.922,-62.771,176.783,16.330,152.125
C03406=1097.963,126.673,-62.751,176.780,16.330,152.126
C03407=1097.958,126.423,-62.731,176.777,16.330,152.127
C03408=1097.952,126.174,-62.712,176.774,16.330,152.127
C03409=1097.946,125.925,-62.692,176.771,16.330,152.128
C03410=1097.941,125.675,-62.672,176.768,16.329,152.128
C03411=1097.935,125.426,-62.653,176.766,16.329,152.129
C03412=1097.929,125.177,-62.633,176.762,16.329,152.129
C03413=1097.923,124.928,-62.614,176.759,16.328,152.130
C03414=1097.918,124.680,-62.594,176.757,16.328,152.130
C03415=1097.912,124.430,-62.575,176.754,16.328,152.131
C03416=1097.907,124.181,-62.556,176.751,16.328,152.131
C03417=1097.902,123.931,-62.536,176.748,16.327,152.132
C03418=1097.896,123.682,-62.516,176.745,16.327,152.133
C03419=1097.890,123.433,-62.497,176.743,16.327,152.133
C03420=1097.884,123.183,-62.478,176.739,16.326,152.134
C03421=1097.878,122.934,-62.458,176.737,16.327,152.134
C03422=1097.873,122.686,-62.439,176.734,16.326,152.135
C03423=1097.867,122.436,-62.420,176.731,16.325,152.135
C03424=1097.862,122.187,-62.400,176.728,16.326,152.136
C03425=1097.856,121.938,-62.380,176.725,16.325,152.136
C03426=1097.850,121.689,-62.361,176.722,16.324,152.137
C03427=1097.845,121.440,-62.342,176.719,16.325,152.137
C03428=1097.839,121.190,-62.323,176.716,16.324,152.138
C03429=1097.834,120.941,-62.304,176.714,16.324,152.138
C03430=1097.828,120.692,-62.284,176.711,16.324,152.139
C03431=1097.822,120.443,-62.265,176.708,16.323,152.139
C03432=1097.817,120.194,-62.246,176.705,16.323,152.140
C03433=1097.811,119.945,-62.226,176.702,16.323,152.140
C03434=1097.805,119.695,-62.207,176.700,16.322,152.141
C03435=1097.800,119.446,-62.188,176.696,16.322,152.141
C03436=1097.794,119.196,-62.169,176.694,16.321,152.142
C03437=1097.789,118.948,-62.149,176.691,16.321,152.142
C03438=1097.783,118.699,-62.130,176.688,16.320,152.143
C03439=1097.777,118.449,-62.111,176.686,16.321,152.143
C03440=1097.772,118.200,-62.091,176.682,16.320,152.144
C03441=1097.767,117.951,-62.073,176.679,16.319,152.144
C03442=1097.761,117.702,-62.053,176.677,16.320,152.145
C03443=1097.755,117.452,-62.034,176.674,16.319,152.145
C03444=1097.749,117.203,-62.015,176.671,16.319,152.146
C03445=1097.744,116.954,-61.996,176.668,16.318,152.146
C03446=1097.739,116.705,-61.977,176.665,16.318,152.147
C03447=1097.733,116.455,-61.957,176.663,16.317,152.147
C03448=1097.728,116.206,-61.939,176.660,16.317,152.148
C03449=1097.722,115.957,-61.919,176.657,16.316,152.148
C03450=1097.717,115.708,-61.900,176.655,16.316,152.149
C03451=1097.711,115.459,-61.881,176.651,16.316,152.149
C03452=1097.706,115.209,-61.862,176.649,16.315,152.150
C03453=1097.700,114.960,-61.843,176.646,16.315,152.150
C03454=1097.694,114.712,-61.824,176.643,16.314,152.151
C03455=1097.689,114.462,-61.805,176.640,16.314,152.151
C03456=1097.683,114.213,-61.786,176.637,16.314,152.152
C03457=1097.677,113.963,-61.767,176.635,16.314,152.152
C03458=1097.672,113.714,-61.749,176.632,16.313,152.153
C03459=1097.666,113.465,-61.730,176.630,16.313,152.153
C03460=1097.660,113.215,-61.711,176.627,16.312,152.154
C03461=1097.655,112.967,-61.692,176.624,16.311,152.154
C03462=1097.650,112.717,-61.673,176.621,16.312,152.155
C03463=1097.643,112.468,-61.654,176.618,16.311,152.155
C03464=1097.638,112.194,-61.633,176.615,16.310,152.156
C03465=1097.631,111.919,-61.612,176.612,16.311,152.156
C03466=1097.625,111.644,-61.592,176.609,16.310,152.157
C03467=1097.618,111.370,-61.571,176.606,16.309,152.157
C03468=1097.613,111.121,-61.552,176.603,16.309,152.158
C03469=1097.607,110.872,-61.533,176.601,16.309,152.158
C03470=1097.602,110.622,-61.515,176.598,16.308,152.159
C03471=1097.596,110.373,-61.496,176.595,16.308,152.159
C03472=1097.590,110.124,-61.477,176.592,16.307,152.160
C03473=1097.584,109.875,-61.458,176.589,16.307,152.160
C03474=1097.580,109.625,-61.440,176.587,16.307,152.161
C03475=1097.573,109.376,-61.421,176.584,16.306,152.161
C03476=1097.567,109.127,-61.402,176.581,16.306,152.161
C03477=1097.562,108.878,-61.383,176.578,16.305,152.162
C03478=1097.556,108.628,-61.365,176.575,16.304,152.162
C03479=1097.551,108.379,-61.346,176.573,16.305,152.163
C03480=1097.545,108.130,-61.327,176.570,16.304,152.163
C03481=1097.539,107.880,-61.309,176.568,16.304,152.164
C03482=1097.534,107.632,-61.290,176.565,16.303,152.164
C03483=1097.528,107.383,-61.271,176.562,16.303,152.165
C03484=1097.522,107.132,-61.253,176.559,16.302,152.165
C03485=1097.517,106.884,-61.235,176.556,16.302,152.166
C03486=1097.511,106.635,-61.215,176.554,16.302,152.166
C03487=1097.505,106.385,-61.197,176.551,16.301,152.167
C03488=1097.500,106.136,-61.179,176.549,16.300,152.167
C03489=1097.494,105.887,-61.159,176.546,16.300,152.168
C03490=1097.488,105.638,-61.142,176.543,16.300,152.168
C03491=1097.483,105.388,-61.122,176.540,16.299,152.168
C03492=1097.477,105.139,-61.105,176.538,16.299,152.169
C03493=1097.472,104.890,-61.086,176.535,16.298,152.169
C03494=1097.465,104.641,-61.067,176.532,16.298,152.170
C03495=1097.460,104.391,-61.049,176.530,16.297,152.170
C03496=1097.454,104.142,-61.030,176.527,16.296,152.171
C03497=1097.449,103.893,-61.012,176.525,16.296,152.171
C03498=1097.443,103.644,-60.993,176.521,16.296,152.172
C03499=1097.438,103.394,-60.975,176.519,16.296,152.172
C03500=1097.432,103.145,-60.957,176.516,16.295,152.172
C03501=1097.427,102.896,-60.938,176.513,16.294,152.173
C03502=1097.421,102.646,-60.919,176.511,16.294,152.173
C03503=1097.416,102.397,-60.902,176.508,16.293,152.174
C03504=1097.410,102.148,-60.882,176.506,16.293,152.174
C03505=1097.404,101.899,-60.865,176.503,16.292,152.175
C03506=1097.399,101.649,-60.846,176.500,16.292,152.175
C03507=1097.393,101.400,-60.828,176.497,16.291,152.175
C03508=1097.387,101.151,-60.810,176.495,16.291,152.176
C03509=1097.382,100.902,-60.791,176.492,16.290,152.176
C03510=1097.376,100.652,-60.773,176.489,16.289,152.177
C03511=1097.370,100.404,-60.755,176.487,16.289,152.177
C03512=1097.365,100.154,-60.736,176.484,16.289,152.178
C03513=1097.359,99.905,-60.719,176.482,16.288,152.178
C03514=1097.353,99.656,-60.700,176.479,16.288,152.179
C03515=1097.348,99.406,-60.682,176.477,16.287,152.179
C03516=1097.342,99.157,-60.664,176.474,16.287,152.179
C03517=1097.336,98.908,-60.646,176.471,16.286,152.180
C03518=1097.331,98.658,-60.627,176.468,16.285,152.180
C03519=1097.325,98.409,-60.610,176.466,16.285,152.181
C03520=1097.319,98.160,-60.591,176.463,16.285,152.181
C03521=1097.314,97.911,-60.573,176.460,16.284,152.182
C03522=1097.308,97.661,-60.555,176.458,16.284,152.182
C03523=1097.302,97.412,-60.537,176.455,16.283,152.182
C03524=1097.297,97.162,-60.518,176.453,16.283,152.183
C03525=1097.291,96.913,-60.501,176.450,16.282,152.183
C03526=1097.285,96.664,-60.482,176.447,16.282,152.184
C03527=1097.279,96.415,-60.464,176.445,16.281,152.184
C03528=1097.273,96.141,-60.445,176.442,16.280,152.185
C03529=1097.267,95.866,-60.424,176.439,16.280,152.185
C03530=1097.261,95.592,-60.404,176.436,16.279,152.186
C03531=1097.254,95.316,-60.385,176.433,16.279,152.186
C03532=1097.249,95.068,-60.367,176.430,16.278,152.186
C03533=1097.243,94.819,-60.349,176.428,16.277,152.187
C03534=1097.238,94.569,-60.331,176.425,16.277,152.187
C03535=1097.232,94.320,-60.313,176.423,16.276,152.188
C03536=1097.226,94.070,-60.295,176.420,16.276,152.188
C03537=1097.220,93.821,-60.277,176.418,16.275,152.188
C03538=1097.215,93.572,-60.259,176.415,16.274,152.189
C03539=1097.209,93.323,-60.241,176.413,16.274,152.189
C03540=1097.204,93.074,-60.223,176.410,16.273,152.190
C03541=1097.198,92.824,-60.206,176.408,16.273,152.190
C03542=1097.192,92.575,-60.188,176.405,16.272,152.190
C03543=1097.187,92.325,-60.169,176.402,16.272,152.191
C03544=1097.181,92.076,-60.151,176.399,16.271,152.191
C03545=1097.176,91.827,-60.134,176.397,16.271,152.192
C03546=1097.170,91.578,-60.116,176.394,16.270,152.192
C03547=1097.164,91.328,-60.098,176.392,16.268,152.192
C03548=1097.159,91.079,-60.080,176.389,16.268,152.193
C03549=1097.153,90.830,-60.062,176.386,16.267,152.193
C03550=1097.147,90.580,-60.044,176.384,16.267,152.194
C03551=1097.142,90.331,-60.026,176.381,16.266,152.194
C03552=1097.136,90.082,-60.009,176.379,16.266,152.194
C03553=1097.130,89.832,-59.991,176.376,16.265,152.195
C03554=1097.125,89.583,-59.973,176.374,16.265,152.195
C03555=1097.119,89.334,-59.955,176.371,16.264,152.196
C03556=1097.113,89.085,-59.938,176.369,16.264,152.196
C03557=1097.108,88.836,-59.920,176.366,16.263,152.196
C03558=1097.101,88.586,-59.902,176.364,16.262,152.197
C03559=1097.096,88.337,-59.885,176.361,16.262,152.197
C03560=1097.090,88.088,-59.867,176.359,16.261,152.198
C03561=1097.085,87.837,-59.850,176.356,16.261,152.198
C03562=1097.079,87.588,-59.832,176.354,16.260,152.198
C03563=1097.074,87.339,-59.815,176.351,16.259,152.199
C03564=1097.067,87.090,-59.797,176.349,16.259,152.199
C03565=1097.062,86.841,-59.779,176.346,16.258,152.200
C03566=1097.056,86.592,-59.762,176.344,16.258,152.200
C03567=1097.051,86.343,-59.744,176.341,16.257,152.200
C03568=1097.045,86.093,-59.726,176.339,16.256,152.201
C03569=1097.039,85.844,-59.709,176.336,16.255,152.201
C03570=1097.034,85.595,-59.691,176.334,16.255,152.201
C03571=1097.028,85.344,-59.674,176.331,16.254,152.202
C03572=1097.022,85.095,-59.656,176.329,16.254,152.202
C03573=1097.017,84.846,-59.639,176.326,16.253,152.203
C03574=1097.011,84.597,-59.621,176.324,16.253,152.203
C03575=1097.005,84.347,-59.603,176.321,16.252,152.203
C03576=1097.000,84.098,-59.587,176.319,16.251,152.204
C03577=1096.994,83.849,-59.570,176.316,16.250,152.204
C03578=1096.988,83.600,-59.552,176.314,16.250,152.204
C03579=1096.982,83.350,-59.534,176.311,16.249,152.205
C03580=1096.977,83.101,-59.516,176.309,16.248,152.205
C03581=1096.971,82.852,-59.500,176.306,16.248,152.206
C03582=1096.966,82.603,-59.482,176.304,16.247,152.206
C03583=1096.960,82.353,-59.464,176.301,16.246,152.206
C03584=1096.954,82.103,-59.447,176.299,16.246,152.207
C03585=1096.949,81.854,-59.430,176.296,16.245,152.207
C03586=1096.943,81.605,-59.412,176.294,16.244,152.207
C03587=1096.938,81.356,-59.395,176.291,16.244,152.208
C03588=1096.931,81.106,-59.378,176.289,16.243,152.208
C03589=1096.926,80.857,-59.360,176.286,16.242,152.208
C03590=1096.920,80.608,-59.343,176.284,16.242,152.209
C03591=1096.915,80.358,-59.326,176.281,16.240,152.209
C03592=1096.909,80.084,-59.306,176.278,16.240,152.210
C03593=1096.903,79.810,-59.288,176.276,16.239,152.210
C03594=1096.896,79.535,-59.269,176.273,16.238,152.210
C03595=1096.890,79.261,-59.249,176.270,16.237,152.211
C03596=1096.885,79.011,-59.232,176.268,16.237,152.211
C03597=1096.879,78.762,-59.215,176.265,16.236,152.211
C03598=1096.873,78.512,-59.198,176.263,16.236,152.212
C03599=1096.868,78.263,-59.180,176.260,16.235,152.212
C03600=1096.862,78.014,-59.163,176.258,16.234,152.212
C03601=1096.856,77.765,-59.147,176.255,16.233,152.213
C03602=1096.851,77.516,-59.129,176.253,16.233,152.213
C03603=1096.845,77.266,-59.112,176.250,16.232,152.214
C03604=1096.839,77.016,-59.094,176.249,16.231,152.214
C03605=1096.833,76.767,-59.078,176.246,16.230,152.214
C03606=1096.828,76.518,-59.060,176.243,16.230,152.215
C03607=1096.823,76.268,-59.044,176.241,16.229,152.215
C03608=1096.816,76.019,-59.027,176.239,16.228,152.215
C03609=1096.811,75.770,-59.010,176.236,16.227,152.216
C03610=1096.805,75.520,-58.992,176.234,16.227,152.216
C03611=1096.799,75.271,-58.976,176.231,16.226,152.216
C03612=1096.794,75.022,-58.958,176.229,16.225,152.217
C03613=1096.788,74.772,-58.941,176.226,16.224,152.217
C03614=1096.782,74.523,-58.924,176.224,16.224,152.217
C03615=1096.777,74.274,-58.907,176.221,16.223,152.218
C03616=1096.771,74.025,-58.890,176.219,16.222,152.218
C03617=1096.765,73.775,-58.874,176.216,16.221,152.218
C03618=1096.759,73.526,-58.856,176.214,16.221,152.219
C03619=1096.753,73.276,-58.839,176.212,16.220,152.219
C03620=1096.748,73.026,-58.823,176.209,16.219,152.219
C03621=1096.743,72.777,-58.805,176.207,16.219,152.220
C03622=1096.737,72.528,-58.789,176.204,16.218,152.220
C03623=1096.732,72.278,-58.772,176.203,16.217,152.220
